//
CASE stCommand.PositionType OF
	DUT_Command_PositionType.AbsolutePosition:
		F_AddElement(_Command, _Delimiter, _ChangeTypeA);
	DUT_Command_PositionType.RelativePosition:
		F_AddElement(_Command, _Delimiter, _ChangeTypeR);
END_CASE

//
F_AddElement(_Command, _Delimiter, LREAL_TO_STRING(stCommand.Speed));

//
CASE stCommand.CoordSystem OF
	SMC_COORD_SYSTEM.ACS:
		F_AddElement(_Command, _Delimiter, _CoordSystemAcs);
	SMC_COORD_SYSTEM.MCS:
		F_AddElement(_Command, _Delimiter, _CoordSystemMcs);
	SMC_COORD_SYSTEM.PCS_1:
		F_AddElement(_Command, _Delimiter, _CoordSystemPc1);
	SMC_COORD_SYSTEM.PCS_2:
		F_AddElement(_Command, _Delimiter, _CoordSystemPc2);
	SMC_COORD_SYSTEM.TCS:
		F_AddElement(_Command, _Delimiter, _CoordSystemTcs);
	SMC_COORD_SYSTEM.WCS:
		F_AddElement(_Command, _Delimiter, _CoordSystemWcs);
	SMC_COORD_SYSTEM.ICS:
		F_AddElement(_Command, _Delimiter, _CoordSystemIcs);
END_CASE

//
CASE stCommand.CoordinateType OF
	DUT_Command_CoordinateType.Literal:
		F_AddElement(_Command, _Delimiter, _CoordTypeH);
		F_AddElement(_Command, _Delimiter, LREAL_TO_STRING(stCommand.CoordRef.X));
		F_AddElement(_Command, _Delimiter, LREAL_TO_STRING(stCommand.CoordRef.Y));
		F_AddElement(_Command, _Delimiter, LREAL_TO_STRING(stCommand.CoordRef.Z));
		F_AddElement(_Command, _Delimiter, LREAL_TO_STRING(stCommand.CoordRef.A));
		F_AddElement(_Command, _Delimiter, LREAL_TO_STRING(stCommand.CoordRef.B));
		F_AddElement(_Command, _Delimiter, LREAL_TO_STRING(stCommand.CoordRef.C));
		
	DUT_Command_CoordinateType.Variable:
		F_AddElement(_Command, _Delimiter, _CoordTypeV);
		CASE stCommand.ArrayType OF
			DUT_Command_ArrayType.StoredPosition:
				F_AddElement(_Command, _Delimiter, _ArrayTypeS);
			DUT_Command_ArrayType.VisionRegister:
				F_AddElement(_Command, _Delimiter, _ArrayTypeV);
			DUT_Command_ArrayType.Flag:
				// on damn
		END_CASE
		F_AddElement(_Command, _Delimiter, UDINT_TO_STRING(stCommand.ArrayIndex));
		
END_CASE

// only add if move type is circle
IF stCommand.MoveType = DUT_Command_MoveType.CircularMove THEN
	//
	CASE stCommand.CircleMode OF
		SMC_CIRC_MODE.BORDER:
			F_AddElement(_Command, _Delimiter, _CircleModeBor);
		SMC_CIRC_MODE.CENTER:
			F_AddElement(_Command, _Delimiter, _CircleModeCen);
		SMC_CIRC_MODE.RADIUS:
			F_AddElement(_Command, _Delimiter, _CircleModeRad);
	END_CASE
	//
	CASE stCommand.PathChoice OF
		MC_CIRC_PATHCHOICE.CLOCKWISE:
			F_AddElement(_Command, _Delimiter, _PathChoiceClw);
		MC_CIRC_PATHCHOICE.COUNTER_CLOCKWISE:
			F_AddElement(_Command, _Delimiter, _PathChoiceCcw);
	END_CASE
	//
	CASE stCommand.CircularCoordinateType OF
		DUT_Command_CoordinateType.Literal:
			F_AddElement(_Command, _Delimiter, _CoordTypeH);
			F_AddElement(_Command, _Delimiter, LREAL_TO_STRING(stCommand.CoordRef2.X));
			F_AddElement(_Command, _Delimiter, LREAL_TO_STRING(stCommand.CoordRef2.Y));
			F_AddElement(_Command, _Delimiter, LREAL_TO_STRING(stCommand.CoordRef2.Z));
			F_AddElement(_Command, _Delimiter, LREAL_TO_STRING(stCommand.CoordRef2.A));
			F_AddElement(_Command, _Delimiter, LREAL_TO_STRING(stCommand.CoordRef2.B));
			F_AddElement(_Command, _Delimiter, LREAL_TO_STRING(stCommand.CoordRef2.C));
			
		DUT_Command_CoordinateType.Variable:
			F_AddElement(_Command, _Delimiter, _CoordTypeV);
			CASE stCommand.CircularArrayType OF
				DUT_Command_ArrayType.StoredPosition:
					F_AddElement(_Command, _Delimiter, _ArrayTypeS);
				DUT_Command_ArrayType.VisionRegister:
					F_AddElement(_Command, _Delimiter, _ArrayTypeV);
				DUT_Command_ArrayType.Flag:
					// oh damn
			END_CASE
			F_AddElement(_Command, _Delimiter, UDINT_TO_STRING(stCommand.CircularArrayIndex));
			
	END_CASE

END_IF

// set function equal to command
F_BuildMoveCmd := _Command;
                  
END_FUNCTION

FUNCTION F_RoundLreal : LREAL
VAR_INPUT
   rIn : LREAL;      
   Digit: INT;         
END_VAR

VAR
   d1 : DINT;
   r0,r1,r2,Rdigit: LREAL;               
END_VAR

                    // https://forge.codesys.com/forge/talk/Engineering/thread/8d1ee86294/
rdigit   :=INT_TO_LREAL(Digit);
r0 := EXPT(10,rdigit); 
r1 := rIn * r0;
d1 := TRUNC(r1);
r2 := DINT_TO_LREAL(d1);
F_RoundLreal := r2 / r0;
                  
END_FUNCTION

FUNCTION_BLOCK FB_ParseLogicCmd
VAR_INPUT
	Command: STRING(GVL.COMMAND_LEN);
END_VAR
VAR_OUTPUT
	stCommand: ST_LogicCmd;
	Error: BOOL;
	ErrorDescription: STRING;
END_VAR
VAR
	_CmdParams: ARRAY [0..GVL.COMMAND_LEN] OF STRING;
	_i, _j, _k: INT;
END_VAR

                    // IF PASS|INPUT|REGISTER|COUNTER <index> >|<|=|>=|<= <value>
// THEN OUTPUT|JUMP|CALL|CNTUP|CNTDN|CNTRST|REGISTER|NOP <index> <value>
// ELSE OUTPUT|JUMP|CALL|CNTUP|CNTDN|CNTRST|REGISTER|NOP <index> <value>
//
// IF_Condition
// IF_Condition_Idx
// IF_Condition_Operator
// IF_Condition_Operator_Compare
// THEN_Function
// THEN_Function_Value
// THEN_Function_Idx
// ELSE_Function
// ELSE_Function_Idx
// ELSE_Function_Value

Error:=FALSE;
ErrorDescription:='';

// split command string into commands
_CmdParams:=F_SplitCmd(Command:=Command);

//
_i := 0;

// disregard the 'IF'
_i := _i + 1;

//
IF _CmdParams[_i] = TO_STRING(E_LogicIfCondition.PASS) THEN
	stCommand.IF_Condition := E_LogicIfCondition.PASS;
ELSIF  _CmdParams[_i] = TO_STRING(E_LogicIfCondition.INPUT) THEN
	stCommand.IF_Condition := E_LogicIfCondition.INPUT;
ELSIF  _CmdParams[_i] = TO_STRING(E_LogicIfCondition.REGISTER) THEN
	stCommand.IF_Condition := E_LogicIfCondition.REGISTER;
ELSIF  _CmdParams[_i] = TO_STRING(E_LogicIfCondition.COUNTER) THEN
	stCommand.IF_Condition := E_LogicIfCondition.COUNTER;
ELSIF  _CmdParams[_i] = TO_STRING(E_LogicIfCondition.FLAG) THEN
	stCommand.IF_Condition := E_LogicIfCondition.FLAG;
END_IF
_i := _i + 1;

//
IF stCommand.IF_Condition <> E_LogicIfCondition.PASS THEN
	
	//
	stCommand.IF_Condition_Idx := STRING_TO_INT(_CmdParams[_i]);
	_i := _i + 1;
	
	//
	IF _CmdParams[_i] = TO_STRING(E_LogicIfConditionOperator.GRT) THEN
		stCommand.IF_Condition_Operator := E_LogicIfConditionOperator.GRT;
	ELSIF _CmdParams[_i] = TO_STRING(E_LogicIfConditionOperator.LES) THEN
		stCommand.IF_Condition_Operator := E_LogicIfConditionOperator.LES;                   
	ELSIF _CmdParams[_i] = TO_STRING(E_LogicIfConditionOperator.EQU) THEN
		stCommand.IF_Condition_Operator := E_LogicIfConditionOperator.EQU;
	ELSIF _CmdParams[_i] = TO_STRING(E_LogicIfConditionOperator.GRE) THEN
		stCommand.IF_Condition_Operator := E_LogicIfConditionOperator.GRE;
	ELSIF _CmdParams[_i] = TO_STRING(E_LogicIfConditionOperator.LEQ) THEN
		stCommand.IF_Condition_Operator := E_LogicIfConditionOperator.LEQ;
	END_IF
	_i := _i + 1;
	
	//
	stCommand.IF_Condition_Operator_Value := STRING_TO_UDINT(_CmdParams[_i]);
	_i := _i + 1;
	
END_IF

// disregard the 'THEN'
_i := _i + 1;

//
IF _CmdParams[_i] = TO_STRING(E_LogicFunction.OUTPUT) THEN
	stCommand.THEN_Function := E_LogicFunction.OUTPUT;
ELSIF _CmdParams[_i] = TO_STRING(E_LogicFunction.JUMP) THEN
	stCommand.THEN_Function := E_LogicFunction.JUMP;
ELSIF _CmdParams[_i] = TO_STRING(E_LogicFunction.CALL) THEN
	stCommand.THEN_Function := E_LogicFunction.CALL;           
ELSIF _CmdParams[_i] = TO_STRING(E_LogicFunction.CNTUP) THEN
	stCommand.THEN_Function := E_LogicFunction.CNTUP;
ELSIF _CmdParams[_i] = TO_STRING(E_LogicFunction.CNTDN) THEN
	stCommand.THEN_Function := E_LogicFunction.CNTDN;
ELSIF _CmdParams[_i] = TO_STRING(E_LogicFunction.CNTRST) THEN
	stCommand.THEN_Function := E_LogicFunction.CNTRST;
ELSIF _CmdParams[_i] = TO_STRING(E_LogicFunction.REGISTER) THEN
	stCommand.THEN_Function := E_LogicFunction.REGISTER;
ELSIF _CmdParams[_i] = TO_STRING(E_LogicFunction.FLAG) THEN
	stCommand.THEN_Function := E_LogicFunction.FLAG;
ELSIF _CmdParams[_i] = TO_STRING(E_LogicFunction.NOP) THEN
	stCommand.THEN_Function := E_LogicFunction.NOP;
END_IF
_i := _i + 1;

//
IF stCommand.THEN_Function <> E_LogicFunction.NOP THEN
	stCommand.THEN_Function_Idx := STRING_TO_INT(_CmdParams[_i]);
	_i := _i + 1;
	IF stCommand.THEN_Function = E_LogicFunction.OUTPUT OR
		stCommand.THEN_Function = E_LogicFunction.REGISTER OR
		stCommand.THEN_Function = E_LogicFunction.FLAG THEN
			stCommand.THEN_Function_Value := STRING_TO_UDINT(_CmdParams[_i]);
			_i := _i + 1;
	END_IF
END_IF

// disregard the 'ELSE'
_i := _i + 1;

//
IF _CmdParams[_i] = TO_STRING(E_LogicFunction.OUTPUT) THEN
	stCommand.ELSE_Function := E_LogicFunction.OUTPUT;
ELSIF _CmdParams[_i] = TO_STRING(E_LogicFunction.JUMP) THEN
	stCommand.ELSE_Function := E_LogicFunction.JUMP;
ELSIF _CmdParams[_i] = TO_STRING(E_LogicFunction.CALL) THEN
	stCommand.ELSE_Function := E_LogicFunction.CALL;
ELSIF _CmdParams[_i] = TO_STRING(E_LogicFunction.CNTUP) THEN
	stCommand.ELSE_Function := E_LogicFunction.CNTUP;
ELSIF _CmdParams[_i] = TO_STRING(E_LogicFunction.CNTDN) THEN
	stCommand.ELSE_Function := E_LogicFunction.CNTDN;
ELSIF _CmdParams[_i] = TO_STRING(E_LogicFunction.CNTRST) THEN
	stCommand.ELSE_Function := E_LogicFunction.CNTRST;
ELSIF _CmdParams[_i] = TO_STRING(E_LogicFunction.REGISTER) THEN
	stCommand.ELSE_Function := E_LogicFunction.REGISTER;
ELSIF _CmdParams[_i] = TO_STRING(E_LogicFunction.FLAG) THEN
	stCommand.ELSE_Function := E_LogicFunction.FLAG;
ELSIF _CmdParams[_i] = TO_STRING(E_LogicFunction.NOP) THEN
	stCommand.ELSE_Function := E_LogicFunction.NOP;
END_IF
_i := _i + 1;

//
IF stCommand.ELSE_Function <> E_LogicFunction.NOP THEN
	stCommand.ELSE_Function_Idx := STRING_TO_INT(_CmdParams[_i]);
	_i := _i + 1;
	IF stCommand.ELSE_Function = E_LogicFunction.OUTPUT OR
		stCommand.ELSE_Function = E_LogicFunction.REGISTER OR
		stCommand.ELSE_Function = E_LogicFunction.FLAG THEN
			stCommand.ELSE_Function_Value := STRING_TO_UDINT(_CmdParams[_i]);
			_i := _i + 1;
	END_IF
END_IF
                  
END_FUNCTION_BLOCK

FUNCTION F_BuildLogicCmd : STRING(GVL.COMMAND_LEN)
VAR_INPUT
	stCommand: ST_LogicCmd;
END_VAR
VAR
    _Command: STRING(GVL.COMMAND_LEN);
END_VAR
VAR CONSTANT
	_Delimiter: STRING:=' ';
END_VAR

                    // IF PASS|INPUT|REGISTER|COUNTER <index> >|<|=|>=|<= <value>
// THEN OUTPUT|JUMP|CNTUP|CNTDN|CNTRST|REGISTER|NOP <index> <value>
// ELSE OUTPUT|JUMP|CNTUP|CNTDN|CNTRST|REGISTER|NOP <index> <value>
//
// IF_Condition
// IF_Condition_Idx
// IF_Condition_Operator
// IF_Condition_Operator_Compare
// THEN_Function
// THEN_Function_Value
// THEN_Function_Idx
// ELSE_Function
// ELSE_Function_Idx
// ELSE_Function_Value

// clear the command
_Command:='';

// build command
F_AddElement(_Command, _Delimiter, 'IF');
F_AddElement(_Command, _Delimiter, TO_STRING(stCommand.IF_Condition));
IF stCommand.IF_Condition <> E_LogicIfCondition.PASS THEN
	F_AddElement(_Command, _Delimiter, INT_TO_STRING(stCommand.IF_Condition_Idx));
	F_AddElement(_Command, _Delimiter, TO_STRING(stCommand.IF_Condition_Operator));
	F_AddElement(_Command, _Delimiter, UDINT_TO_STRING(stCommand.IF_Condition_Operator_Value));
END_IF
F_AddElement(_Command, _Delimiter, 'THEN');
F_AddElement(_Command, _Delimiter, TO_STRING(stCommand.THEN_Function));
IF stCommand.THEN_Function <> E_LogicFunction.NOP THEN
	F_AddElement(_Command, _Delimiter, INT_TO_STRING(stCommand.THEN_Function_Idx));
	IF stCommand.THEN_Function = E_LogicFunction.OUTPUT OR 
		stCommand.THEN_Function = E_LogicFunction.REGISTER OR 
		stCommand.THEN_Function = E_LogicFunction.FLAG THEN
			F_AddElement(_Command, _Delimiter, UDINT_TO_STRING(stCommand.THEN_Function_Value));
	END_IF
END_IF
IF stCommand.IF_Condition <> E_LogicIfCondition.PASS THEN
	F_AddElement(_Command, _Delimiter, 'ELSE');
	F_AddElement(_Command, _Delimiter, TO_STRING(stCommand.ELSE_Function));
	IF stCommand.ELSE_Function <> E_LogicFunction.NOP THEN
		F_AddElement(_Command, _Delimiter, INT_TO_STRING(stCommand.ELSE_Function_Idx));
		IF stCommand.ELSE_Function = E_LogicFunction.OUTPUT OR
			stCommand.ELSE_Function = E_LogicFunction.REGISTER OR
			stCommand.ELSE_Function = E_LogicFunction.FLAG THEN
				F_AddElement(_Command, _Delimiter, UDINT_TO_STRING(stCommand.ELSE_Function_Value));
		END_IF
	END_IF
END_IF

// set function equal to command
F_BuildLogicCmd := _Command;
                  
END_FUNCTION

FUNCTION F_HomeOffsetCalc : LREAL
VAR_INPUT
	CurrentOffset: LREAL;
	CurrentPosition: LREAL;
	HomeSearchDirection: MC_Direction;
END_VAR
VAR
END_VAR

                    IF HomeSearchDirection = MC_Direction.positive THEN
	F_HomeOffsetCalc := -F_RoundLreal(ABS(CurrentPosition - CurrentOffset),2);
	
ELSIF HomeSearchDirection = MC_Direction.negative THEN
	F_HomeOffsetCalc := F_RoundLreal(ABS(CurrentPosition - CurrentOffset),2);
	
ELSE
	F_HomeOffsetCalc := CurrentOffset;
	
END_IF
                  
END_FUNCTION

FUNCTION_BLOCK FB_ProgramProcessor EXTENDS FB_Module
VAR_IN_OUT
	Programs: ARRAY [GVL.PROG_ARR_BEG..GVL.PROG_ARR_END] OF DUT_Program;
	J1, J2, J3, J4, J5, J6: AXIS_REF_SM3;
	AxisGroup: AXIS_GROUP_REF_SM3;
	GroupHandler: FB_GroupHandler;
	CmdIO: ST_LogicCmdIO;
END_VAR
VAR_INPUT
	Enable: BOOL;
END_VAR
VAR_OUTPUT
	ItfActiveProcessorUnitMode	: PACK_ML.IUnitMode;
	ItfActiveModule: ItfModule;
	StatusText: STRING(255);
    GCodeLines: ARRAY[0..SMC_GCodeViewer.c_uiLines] OF STRING;
END_VAR
VAR
	_DummyUnitMode: PACK_ML.UnitMode;
	_UnitModeCurrentState: PACK_ML.State;
	_Returning:  ARRAY [GVL.PROG_ARR_BEG..GVL.PROG_ARR_END] OF BOOL;
	_ReturnPrograms: ARRAY [GVL.PROG_ARR_BEG..GVL.PROG_ARR_END] OF UINT;
	_ReturnCommands: ARRAY [GVL.PROG_CMDS_ARR_BEG..GVL.PROG_CMDS_ARR_END + 1] OF UINT; // +1 because we want to be able to tell if calling program was on last command
	_CurrentPrgIdx: UINT;
	_ProcessCommands: FB_CommandProcessor;
	_Commands: ARRAY [GVL.PROG_CMDS_ARR_BEG..GVL.PROG_CMDS_ARR_END] OF DUT_Command;
    _ErrorRtrig: R_TRIG;
	_i, _j, _k: INT;
	_FirstScan: BOOL:=TRUE;
END_VAR

VAR CONSTANT
	_STEP_DONE: 			INT := 1000;
	_STEP_IDLE: 			INT := 0000;
	_STEP_PRG:				INT := 0010;
	_STEP_WAIT_EXECUTE:		INT := 0020;
	_STEP_WAIT_IDLE:		INT := 0025;
	_STEP_ERR:              INT := 0030;
END_VAR

                    //
SUPER^();

//
IF _FirstScan THEN
	// will exception if we don't set this on first scan
	_DummyUnitMode(sName := 'Active Processor', 
					eInitialState := PACK_ML.State.Idle,
					xActive := TRUE);
	ItfActiveProcessorUnitMode := _DummyUnitMode;
END_IF

// this is at best a hack and needs to be rethought out.
// we logically cant assign a process as the active unit mode 
// at start up so we use this dummy one
CASE _DummyUnitMode.CurrentState OF
	PACK_ML.State.Stopped,
	PACK_ML.State.Aborted,
	PACK_ML.State.Held,
	PACK_ML.State.Suspended,
	PACK_ML.State.Complete,
	PACK_ML.State.Idle:
		//
	PACK_ML.State.Resetting,
	PACK_ML.State.Starting,
	PACK_ML.State.Execute,
	PACK_ML.State.Suspending,
	PACK_ML.State.UnSuspending,
	PACK_ML.State.Holding,
	PACK_ML.State.UnHolding,
	PACK_ML.State.Completing,
	PACK_ML.State.Aborting,
	PACK_ML.State.Stopping,
	PACK_ML.State.Clearing:
		_DummyUnitMode.ActingStateCompleted();
END_CASE

// PackML state machine implementation
_UnitModeCurrentState := SUPER^._UnitMode.CurrentState;

//
_ErrorRtrig(CLK:=_ProcessCommands.Error);
IF _ErrorRtrig.Q THEN
	SUPER^.M_Error(Description:=CONCAT('Command Processor Error: ', _ProcessCommands.ErrorDescription));
	StatusText:=SUPER^.ErrorDescription;
END_IF

//
_ProcessCommands(
	StoredPositions:=SUPER^.StoredPositions,
	VisionRegisters:=SUPER^.VisionRegisters,
	Flags:=SUPER^.Flags,
	J1:=J1, J2:=J2, J3:=J3, J4:=J4, J5:=J5, J6:=J6,
	AxisGroup:= AxisGroup,
	GroupHandler:= GroupHandler,
	CmdIO:=CmdIO,
	PrgProcessor:= THIS^,
    GCodeLines => GCodeLines,
	Enable:= Enable,
	Error=> ,
	StatusText=>StatusText);	

_FirstScan := FALSE;
                  

METHOD PUBLIC M_CallProgram : bool
VAR_INPUT
	ProgramNumber: UINT; // program to call
	ReturnProgram: UINT; // number of the program to return to when the call program ends
	ReturnCommand: UINT; // number of the command to start from when called program ends
END_VAR
                          {warning disable C0371}
IF ProgramNumber <= GVL.PROG_ARR_END AND_THEN ProgramNumber >= GVL.PROG_ARR_BEG
	AND_THEN ReturnProgram <= GVL.PROG_ARR_END AND_THEN ReturnProgram >= GVL.PROG_ARR_BEG
	AND_THEN SUPER^.PropCurrentState = PACK_ML.State.Execute THEN
		IF _ProcessCommands.M_SetCommands(StartingCommand:=0, Commands:=Programs[ProgramNumber].Commands) THEN
			IF ReturnCommand <= GVL.PROG_CMDS_ARR_END + 1 AND_THEN ReturnCommand >= GVL.PROG_CMDS_ARR_BEG THEN // +1 because we want to be able to tell if calling program was on last command
				_Returning[ProgramNumber] := TRUE;
				_ReturnPrograms[ProgramNumber] := ReturnProgram;
				_ReturnCommands[ProgramNumber] := ReturnCommand;
			END_IF
			_CurrentPrgIdx := ProgramNumber;
			M_CallProgram := TRUE;
		ELSE
			M_CallProgram := FALSE;
		END_IF
ELSE
	M_CallProgram := FALSE;
END_IF
{warning restore C0371}
                        
END_METHOD

METHOD PROTECTED M_Complete : BOOL
                          // once complete, reset to get back to idle
SUPER^._UnitMode.Reset();
                        
END_METHOD

METHOD PROTECTED M_Resetting : BOOL
                          CASE _SeqResetting OF
	0:
		_ProcessCommands.M_Home();
		_SeqResetting := _SeqResetting + 1;
	1:
		IF _ProcessCommands.PropCurrentState = PACK_ML.State.Idle THEN
			_SeqResetting := 0;
			SUPER^.M_StateComplete();
		END_IF
		
END_CASE

SUPER^.M_Reset();

(*IF ItfActiveModule <> 0 THEN
	CASE _Seq OF
		0:
			IF NOT ItfActiveModule.PropCurrentState = PACK_ML.State.Idle THEN
				ItfActiveModule.M_Home();
				_Seq := 1;
			ELSE
				SUPER^.M_StateComplete();
			END_IF
		1:
			IF ItfActiveModule.PropCurrentState = PACK_ML.State.Idle THEN
				_Seq := 0;
			END_IF
			
	END_CASE
	
ELSE
	SUPER^.M_StateComplete();
	_Seq := 0;
	
END_IF*)
                        
END_METHOD

METHOD PROTECTED M_Idle : BOOL
                          // in this state, we want to reset all the function blocks and hang out
FOR _i:=GVL.PROG_ARR_BEG TO GVL.PROG_ARR_END BY 1 DO
	_Returning[_i] := FALSE;
END_FOR
(*FOR _i:=GVL.PROG_ARR_BEG TO GVL.PROG_ARR_END BY 1 DO
	_ReturnPrograms[_i] := 0;
END_FOR
FOR _i:=GVL.PROG_CMDS_ARR_BEG TO GVL.PROG_CMDS_ARR_END BY 1 DO
	_ReturnCommands[_i] := 0;
END_FOR*)
_SeqMain := _STEP_IDLE;
_SeqAborting := 0;
_SeqClearing := 0;
_SeqResetting := 0;
                        
END_METHOD

METHOD PROTECTED M_SetPackML : BOOL
                          // SUPER already does this but the default is eInitialState:=PACK_ML.State.Idle 
// and we want PACK_ML.State.Aborted for the Orchestrator
SUPER^._UnitMode(sName := 'Program Processor',
				eInitialState := PACK_ML.State.Aborted,
				xActive := TRUE);
                        
END_METHOD

METHOD PROTECTED M_Starting : BOOL
                          // here we want to clear things and get ready for the execute state
// we can consider this the "INIT" state
(*FOR _i:=GVL.PROG_ARR_BEG TO GVL.PROG_ARR_END BY 1 DO
	_Returning[_i] := FALSE;
END_FOR
FOR _i:=GVL.PROG_ARR_BEG TO GVL.PROG_ARR_END BY 1 DO
	_ReturnPrograms[_i] := 0;
END_FOR
FOR _i:=GVL.PROG_CMDS_ARR_BEG TO GVL.PROG_CMDS_ARR_END BY 1 DO
	_ReturnCommands[_i] := 0;
END_FOR*)
//_CurrentPrgIdx := 0;
_SeqMain := _STEP_PRG;
SUPER^.M_StateComplete();
                        
END_METHOD

METHOD PROTECTED M_Execute : BOOL
VAR
    _ErrorDescription: STRING;
END_VAR
                          {warning disable C0371}
// here we want to execute our commands/jobs/etc and set completed when done.
//
CASE _SeqMain OF
  	_STEP_DONE:
		_SeqMain := _STEP_IDLE;
		
	_STEP_IDLE:
		// hang out here until called to run
		_CurrentPrgIdx := 0;
		SUPER^.M_StateComplete();
		
	_STEP_PRG: //
		IF NOT Enable THEN
			_SeqMain := _STEP_DONE;
            IF NOT GVL.Enable THEN
                _ErrorDescription := 'Robot not enabled';
            END_IF
            IF NOT PersistentVars.Flags[GVL.HOME_COMPLETE].Value THEN
                _ErrorDescription := CONCAT(_ErrorDescription, ' | Robot not homed');
            END_IF
            IF GVL.xActiveAlarm THEN
                _ErrorDescription := CONCAT(_ErrorDescription, ' | Active alarms exist');
            END_IF
            IF _ErrorDescription = '' THEN
                _ErrorDescription := 'Not enabled';
            END_IF
            _M_Error(Description := _ErrorDescription);
            
		ELSIF _CurrentPrgIdx <= GVL.PROG_ARR_END AND _CurrentPrgIdx >= GVL.PROG_ARR_BEG THEN
			//
			StatusText := '';
			ItfActiveModule := _ProcessCommands;
			ItfActiveProcessorUnitMode := _ProcessCommands.ItfUnitMode;
			
			IF _ProcessCommands.M_SetCommands(StartingCommand:=0, Commands:=Programs[_CurrentPrgIdx].Commands) THEN
				_ProcessCommands.M_Start();
				_SeqMain := _STEP_WAIT_EXECUTE;
			ELSE
				SUPER^.M_Error('Failed to set Command Processor. Check commands.');
				_SeqMain := _STEP_ERR;
			END_IF
			
				
		ELSE
			_SeqMain := _STEP_DONE;
		END_IF
		
	_STEP_WAIT_EXECUTE:
		IF _ProcessCommands.PropCurrentState = PACK_ML.State.Execute THEN
			_SeqMain := _STEP_WAIT_IDLE;
		END_IF
		
	_STEP_WAIT_IDLE: // wait for program to finish
		//
		IF _ProcessCommands.PropCurrentState = PACK_ML.State.Idle THEN
			IF _Returning[_CurrentPrgIdx] THEN
				_Returning[_CurrentPrgIdx] := FALSE;
				IF _ReturnPrograms[_CurrentPrgIdx] <= GVL.PROG_ARR_END AND_THEN _ReturnPrograms[_CurrentPrgIdx] >= GVL.PROG_ARR_BEG
					AND_THEN _ReturnCommands[_CurrentPrgIdx] <= GVL.PROG_CMDS_ARR_END + 1 AND_THEN _ReturnCommands[_CurrentPrgIdx] >= GVL.PROG_CMDS_ARR_BEG // +1 because we want to be able to tell if calling program was on last command
					THEN
						//
						IF _ProcessCommands.M_SetCommands(StartingCommand:=_ReturnCommands[_CurrentPrgIdx], Commands:=Programs[_ReturnPrograms[_CurrentPrgIdx]].Commands) THEN
							_CurrentPrgIdx := _ReturnPrograms[_CurrentPrgIdx];
							_ProcessCommands.M_Start();
							_SeqMain := _STEP_WAIT_EXECUTE;
						ELSE
							SUPER^.M_Error('Failed to set Command Processor. Check commands.');
							_SeqMain := _STEP_ERR;
						END_IF
				ELSE
					_SeqMain := _STEP_DONE;
				END_IF
			ELSE
				_SeqMain := _STEP_DONE;
			END_IF
		END_IF
		//
		IF _ProcessCommands.PropError THEN
			SUPER^._UnitMode.Suspend();
			_SeqMain := _STEP_ERR;
		END_IF
		
	_STEP_ERR: //
	
END_CASE

// watch for rising edge of idle state. this was done for all processors since 
// the vision processor runs in a separate task and isnt guaranteed to start in the same 
// PLC scan.
//_ProcessorDoneRtrig(clk:=ItfActiveProcessorUnitMode.CurrentState = PACK_ML.State.Idle);
{warning restore C0371}
                        
END_METHOD

METHOD PROTECTED M_Suspending : BOOL
                          IF ItfActiveModule <> 0 THEN
	IF ItfActiveModule.PropCurrentState = PACK_ML.State.Execute THEN
		ItfActiveModule.M_Hold();
		IF ItfActiveModule.PropCurrentState = PACK_ML.State.Held THEN
			SUPER^.M_StateComplete();
		END_IF
	ELSE
		SUPER^.M_StateComplete();
	END_IF
	
ELSE
	SUPER^.M_StateComplete();
	
END_IF
                        
END_METHOD

METHOD PROTECTED M_UnSuspending : BOOL
                          //
IF ItfActiveModule <> 0 THEN
	ItfActiveModule.M_Start();
	IF ItfActiveModule.PropCurrentState = PACK_ML.State.Execute THEN
		SUPER^.M_StateComplete();
	END_IF
	
ELSE
	SUPER^.M_StateComplete();
	
END_IF

//
_SeqMain := _STEP_WAIT_IDLE;
                        
END_METHOD

METHOD PROTECTED M_Holding : BOOL
                          IF ItfActiveModule <> 0 THEN
	ItfActiveModule.M_Hold();
	IF ItfActiveModule.PropCurrentState = PACK_ML.State.Held THEN
		SUPER^.M_StateComplete();
	END_IF
ELSE
	SUPER^.M_StateComplete();
END_IF
                        
END_METHOD

METHOD PROTECTED M_Unholding : BOOL
                          //
IF ItfActiveModule <> 0 THEN
	ItfActiveModule.M_Start();
	IF ItfActiveModule.PropCurrentState = PACK_ML.State.Execute THEN
		SUPER^.M_StateComplete();
	END_IF
	
ELSE
	SUPER^.M_StateComplete();
	
END_IF

//
_SeqMain := _STEP_WAIT_IDLE;
                        
END_METHOD

METHOD PROTECTED M_Aborting : BOOL
                          CASE _SeqAborting OF
	0:
		_ProcessCommands.M_Abort();
		_SeqAborting := _SeqAborting + 1;
	1:
		IF _ProcessCommands.PropCurrentState = PACK_ML.State.Aborted THEN
			_SeqAborting := 0;
			SUPER^.M_StateComplete();
		END_IF
		
END_CASE

(*IF ItfActiveModule <> 0 THEN
	ItfActiveModule.M_Abort();
	IF ItfActiveModule.PropCurrentState = PACK_ML.State.Aborted THEN
		SUPER^.M_StateComplete();
	END_IF
ELSE
	SUPER^.M_StateComplete();
END_IF*)
                        
END_METHOD

METHOD PROTECTED M_Stopping : BOOL
                          IF ItfActiveModule <> 0 THEN
	ItfActiveModule.M_Stop();
	IF ItfActiveModule.PropCurrentState = PACK_ML.State.Idle 
		OR ItfActiveModule.PropCurrentState = PACK_ML.State.Stopped 
		OR ItfActiveModule.PropCurrentState = PACK_ML.State.Aborted 
		OR ItfActiveModule.PropCurrentState = PACK_ML.State.Complete THEN
			SUPER^.M_StateComplete();
	END_IF
	
ELSE
	SUPER^.M_StateComplete();
	
END_IF
                        
END_METHOD

METHOD PROTECTED M_Clearing : BOOL
                          SUPER^.M_StateComplete();

(*IF SUPER^.Flags[GVL.HOME_COMPLETE].Value THEN
	CASE _SeqClearing OF
		0:
			_ProcessMoveCommand.M_Home();
			_SeqClearing := _SeqClearing + 1;
		1:
			IF _ProcessMoveCommand.PropCurrentState = PACK_ML.State.Idle THEN
				_SeqClearing := _SeqClearing + 1;
			END_IF
		2:
			IF NOT _ProcessMoveCommand.Error THEN
				_ProcessMoveCommand.Command := GVL.Pose2;
				_ProcessMoveCommand.M_Start();
				_SeqClearing := _SeqClearing + 1;
			ELSE
				SUPER^._M_Error(Description:='Move processor errored. Please reset and try again');
				_SeqClearing := -1;
			END_IF
		3:
			IF _ProcessMoveCommand.PropCurrentState = PACK_ML.State.Execute THEN
				_SeqClearing := _SeqClearing + 1;
			END_IF
		4:
			IF _ProcessMoveCommand.PropCurrentState = PACK_ML.State.Complete 
				OR _ProcessMoveCommand.PropCurrentState = PACK_ML.State.Stopped 
				OR _ProcessMoveCommand.PropCurrentState = PACK_ML.State.Aborted
				OR _ProcessMoveCommand.PropCurrentState = PACK_ML.State.Idle  THEN
					SUPER^.M_StateComplete();
					_SeqClearing := 0;
			END_IF
	END_CASE
ELSE
	SUPER^._M_Error(Description:='Drives are not homed. Please home and try again');
	_SeqClearing := -1;
END_IF

IF _ProcessMoveCommand.Error THEN
	SUPER^._M_Error(Description:='Move processor in error state. Please reset and try again');
	_SeqClearing := -1;
END_IF
*)

(*
IF ItfActiveModule <> 0 THEN
	//
	CASE _Seq OF
		0:
			IF NOT ItfActiveModule.PropCurrentState = PACK_ML.State.Stopped THEN
				ItfActiveModule.M_Abort();
				_Seq := 1;
			ELSE
				SUPER^.M_StateComplete();
			END_IF
		1:
			CASE ItfActiveModule.PropCurrentState OF
				PACK_ML.State.Aborted:
					ItfActiveModule.Clear();
				PACK_ML.State.Stopped:
					_Seq := 0;
			END_CASE
			
	END_CASE
ELSE
	_Seq := 0;
	SUPER^.M_StateComplete();
END_IF
*)

                        
END_METHOD

METHOD PUBLIC M_SetProgram : BOOL
VAR_INPUT
	ProgramNumber: UINT;
END_VAR
                          IF ProgramNumber >= GVL.PROG_ARR_BEG AND ProgramNumber <= GVL.PROG_ARR_END THEN
	_CurrentPrgIdx := ProgramNumber;
	M_SetProgram := TRUE;
ELSE
	M_SetProgram := FALSE;
END_IF
                        
END_METHOD

METHOD PRIVATE _M_Error
VAR_INPUT
    Description: STRING;
END_VAR
                          SUPER^.M_Error(Description := CONCAT('Program Processor: ', Description));
                        
END_METHOD

{attribute 'monitoring' := 'variable'}
PROPERTY PUBLIC P_CurrentProgram : REFERENCE TO UINT
GET
VAR
END_VAR
                            P_CurrentProgram REF= _CurrentPrgIdx;
                          
END_GET
END_PROPERTY

{attribute 'monitoring' := 'variable'}
PROPERTY PUBLIC P_CurrentCommand : REFERENCE TO DUT_Command
GET
VAR
END_VAR
                            P_CurrentCommand REF= _ProcessCommands.P_CurrentCommand;
                          
END_GET
END_PROPERTY

{attribute 'monitoring' := 'variable'}
PROPERTY PUBLIC P_CurrentCommandIndex : REFERENCE TO UINT
GET
VAR
END_VAR
                            P_CurrentCommandIndex REF= _ProcessCommands.P_CurrentCommandIndex;
                          
END_GET
END_PROPERTY
END_FUNCTION_BLOCK

FUNCTION_BLOCK FB_Controller EXTENDS FB_PythonServerHandler
VAR_INPUT
END_VAR
VAR_OUTPUT
END_VAR
VAR
	Controller: ST_Controller;
	ControllerStates: ARRAY [0..254] OF BYTE;
	ControllerStatesTemp: ARRAY [0..254] OF BYTE;
	ReadStringTemp: STRING(255);
	RecordLast: DINT;
	ReconnectTimer: TON:=(PT:=T#5S);
	
	_SetColor: BOOL;
	_Red: INT:=0;
	_Green: INT:=255;
	_Blue: INT:=0;
	
	_SetMicrophoneState: BOOL;
	_MicrophoneState: BOOL;
	
	_SetPlayerID: BOOL;
	_PlayerID: E_ControllerPlayerID;
	
	_SetBrightness: BOOL;
	_Brightness: E_ControllerBrightness;
	
	_SetMotorIntensity: BOOL;
	_Motor: E_ControllerMotor;
	_MotorIntensity: USINT; // 0-255
	_MotorIntensityDuration: REAL; // ms
	
	_SetTriggerMode: BOOL;
	_TriggerModeTrigger: E_ControllerTrigger;
	_TriggerModeMode: E_ControllerTriggerMode;
	
	_SetTriggerForce: BOOL;
	_TriggerForceTrigger: E_ControllerTrigger;
	_TriggerForceParameter: E_ControllerTriggerForceParameter;
	_TriggerForceIntensity: USINT;
	
	_i, _j, _k: INT;
	FirstScan: BOOL:=TRUE;
END_VAR
VAR CONSTANT
	States: STRING:='states: ';
END_VAR

                    SUPER^();

// copy over controller states when a new message is received
IF SUPER^.P_RecordNumber <> RecordLast THEN
	RecordLast := SUPER^.P_RecordNumber;
	IF FIND(SUPER^.P_RawReadString, States) > 0 THEN // TODO this is getting messy. need to overhaul how this works
		ControllerStatesTemp := SUPER^.P_RawReadByteArray;
		FOR _i:=0 TO UINT_TO_INT(SIZEOF(ControllerStates)) - LEN(States) BY 1 DO
			ControllerStates[_i] := ControllerStatesTemp[_i + LEN(States)];
		END_FOR
		
	END_IF
END_IF

//
_M_EvaluateControllerStates(States:=ControllerStates);
_M_SetColor();
_M_SetMicrophoneState();
_M_SetPlayerID();
_M_SetBrightness();
_M_SetMotorIntensity();
_M_SetTriggerMode();
_M_SetTriggerForce();

// try to reconnect to the server when data stops?
// leave this commented out until we have a better condition
// the edge case is when the controller is connected via bluetooth 
// but for some reason the server is not connected to it.
// maybe work this issue out on the server side.
(*ReconnectTimer(IN:= RecordLast=SUPER^.P_RecordNumber);
IF ReconnectTimer.Q THEN
	ReconnectTimer(IN:=FALSE);
	SUPER^.M_Reconnect();
END_IF*)

FirstScan:=FALSE;
                  

METHOD PRIVATE _M_EvaluateControllerStates : BOOL
VAR_INPUT
	States: ARRAY[0..254] OF BYTE;
END_VAR
VAR_STAT
	_i, _j, _k: UINT;
	_FirstScan: BOOL:=TRUE;
	_HeartbeatTimer: TON:=(PT:=T#2S);
	_Heartbeat: USINT:=0;
	_HeartbeatLast: USINT:=0;
END_VAR
VAR CONSTANT
END_VAR
                          IF _FirstScan THEN
	//
END_IF

//
_Heartbeat := States[0] OR States[7]; // States[0] appears to be bluetooth and States[7] appears to be wired
IF _Heartbeat <> _HeartbeatLast THEN
	_HeartbeatLast := _Heartbeat;
	_HeartbeatTimer(IN:=FALSE);
ELSE
	_HeartbeatTimer(IN:=TRUE);
END_IF
Controller.Connected S= NOT _HeartbeatTimer.IN;
Controller.Connected R= _HeartbeatTimer.Q;

// clear all the data if the controller disconnects
IF NOT Controller.Connected THEN
	//MemUtils.MemSet(pbyBuffer:=ADR(States), byValue:=0, dwSize:=SIZEOF(States)); 
	FOR _i:=1 TO 254 BY 1 DO // start at 1 so we dont overwrite the heartbeat
		States[_i] := 0;
	END_FOR
END_IF

Controller.Joysticks.Left.X					:= States[1];
Controller.Joysticks.Left.Y					:= States[2];
Controller.Joysticks.Right.X				:= States[3];
Controller.Joysticks.Right.Y				:= States[4];
Controller.Triggers.Left.Two				:= States[5];
Controller.Triggers.Right.Two				:= States[6];

//UNUSED									:= States[7];

Controller.Buttons.Triangle 				:= States[8].7;
Controller.Buttons.Circle 					:= States[8].6;
Controller.Buttons.Cross 					:= States[8].5;
Controller.Buttons.Square 					:= States[8].4;
Controller.Dpad								:= F_DpadState(States[8] AND 16#0F);

Controller.Joysticks.Right.ThreeButton 		:= States[9].7;
Controller.Joysticks.Left.ThreeButton 		:= States[9].6;
Controller.Buttons.Options 					:= States[9].5;
Controller.Buttons.Share 					:= States[9].4;
Controller.Triggers.Right.TwoButton 		:= States[9].3;
Controller.Triggers.Left.TwoButton 			:= States[9].2;
Controller.Triggers.Right.One 				:= States[9].1;
Controller.Triggers.Left.One 				:= States[9].0;

Controller.Buttons.PS						:= States[10].0;
Controller.Buttons.Touch					:= States[10].1;
Controller.Buttons.Mic						:= States[10].2;

//UNUSED									:= States[11];
//UNUSED									:= States[12];
//UNUSED									:= States[13];
//UNUSED									:= States[14];
//UNUSED									:= States[15];

{warning disable C0308}
Controller.Accelerometer.X					:= SHL(States[16], 8) OR States[17];
Controller.Accelerometer.Y					:= SHL(States[18], 8) OR States[19];
Controller.Accelerometer.Z					:= SHL(States[20], 8) OR States[21];

Controller.Gyroscope.Pitch					:= SHL(States[22], 8) OR States[23];
Controller.Gyroscope.Yaw					:= SHL(States[24], 8) OR States[25];
Controller.Gyroscope.Roll					:= SHL(States[26], 8) OR States[27];

//UNUSED									:= States[28];
//UNUSED									:= States[29];
//UNUSED									:= States[30];
//UNUSED									:= States[31];
//UNUSED									:= States[32];

Controller.Trackpads.One.ID					:= States[33] AND 16#7F;
Controller.Trackpads.One.Active				:= (States[33] AND 16#80) = 0;
Controller.Trackpads.One.X					:= SHL((States[35] AND 16#0F), 8) OR States[34];
Controller.Trackpads.One.Y					:= SHL(States[36], 4) OR SHR((States[35] AND 16#F0), 4);
Controller.Trackpads.Two.ID					:= States[37] AND 16#7F;
Controller.Trackpads.Two.Active				:= (States[37] AND 16#80) = 0;
Controller.Trackpads.Two.X					:= SHL((States[39] AND 16#0F), 8) OR States[38];
Controller.Trackpads.Two.Y					:= SHL(States[40], 4) OR SHR((States[39] AND 16#F0), 4);
{warning restore C0308}

//UNUSED									:= States[41];
//UNUSED									:= States[42];
//UNUSED									:= States[43];
//UNUSED									:= States[44];
//UNUSED									:= States[45];
//UNUSED									:= States[46];
//UNUSED									:= States[47];
//UNUSED									:= States[48];
//UNUSED									:= States[49];
//UNUSED									:= States[50];
//UNUSED									:= States[51];
//UNUSED									:= States[52];

// from kit-nya
Controller.Battery.State					:= SHR(States[53] AND 16#F0, 4);
Controller.Battery.Level					:= MIN((States[53] AND 16#0F) * 10 + 5, 100); // TODO this will show a value of 5 when controller is disconnected.

// dont put anything below this
_FirstScan := FALSE;
                        
END_METHOD

METHOD PUBLIC M_SetColor : BOOL
VAR_INPUT
	Red: INT:=0;
	Green: INT:=255;
	Blue: INT:=0;
END_VAR
                          IF Red>=0 AND_THEN Red<=255
	AND_THEN Green>=0 AND_THEN Green<=255
	AND_THEN Blue>=0 AND_THEN Blue<=255THEN
		M_SetColor := TRUE;
		_SetColor:=TRUE;
		_Red:=Red;
		_Green:=Green;
		_Blue:=Blue;
ELSE
	M_SetColor := FALSE;
END_IF
                        
END_METHOD

METHOD PUBLIC M_SetPlayerID : BOOL
VAR_INPUT
	PlayerID: E_ControllerPlayerID;
END_VAR
                          M_SetPlayerID := TRUE;
_PlayerID := PlayerID;
_SetPlayerID := TRUE;

                        
END_METHOD

METHOD PUBLIC M_SetMicrophoneState : BOOL
VAR_INPUT
	State: BOOL;
END_VAR
                          M_SetMicrophoneState := TRUE;
_MicrophoneState := State;
_SetMicrophoneState := TRUE;
                        
END_METHOD

METHOD PRIVATE _M_SetColor : BOOL
VAR_INPUT
END_VAR
VAR
	_Command: STRING(255);
END_VAR
                          IF NOT SUPER^._Busy AND_THEN _SetColor THEN
	_SetColor := FALSE;
	
	_Command := CONCAT('cmd: setColorI:', INT_TO_STRING(_Red));
	_Command := CONCAT(_Command, ',');
	_Command := CONCAT(_Command, INT_TO_STRING(_Green));
	_Command := CONCAT(_Command, ',');
	_Command := CONCAT(_Command, INT_TO_STRING(_Blue));
	
	SUPER^._M_Execute(Command:=_Command, Timeout:=5);
	SUPER^(); // call super here so other methods see it busy.
END_IF
                        
END_METHOD

METHOD PRIVATE _M_SetMicrophoneState : BOOL
VAR_INPUT
END_VAR
VAR
	_Command: STRING(255);
END_VAR
                          IF NOT SUPER^._Busy AND _SetMicrophoneState THEN
	_SetMicrophoneState := FALSE;
	
	_Command := CONCAT('cmd: setMicrophoneState:', BOOL_TO_STRING(_MicrophoneState));
	
	SUPER^._M_Execute(Command:=_Command, Timeout:=5);
	SUPER^(); // call super here so other methods see it busy.
END_IF;
                        
END_METHOD

METHOD PRIVATE _M_SetPlayerID : BOOL
VAR_INPUT
END_VAR
VAR
	_Command: STRING(255);
END_VAR
                          IF NOT SUPER^._Busy AND _SetPlayerID THEN
	_SetPlayerID := FALSE;
	
	_Command := CONCAT('cmd: setPlayerID:', INT_TO_STRING(_PlayerID));
	
	SUPER^._M_Execute(Command:=_Command, Timeout:=5);
	SUPER^(); // call super here so other methods see it busy.
END_IF
                        
END_METHOD

METHOD PRIVATE _M_SetBrightness : BOOL
VAR_INPUT
END_VAR
                          IF NOT SUPER^._Busy AND _SetBrightness THEN
	_SetBrightness := FALSE;
	
	_Command := CONCAT('cmd: setBrightness:', INT_TO_STRING(_Brightness));
	
	SUPER^._M_Execute(Command:=_Command, Timeout:=5);
	SUPER^(); // call super here so other methods see it busy.
END_IF
                        
END_METHOD

METHOD PUBLIC M_SetBrightness : BOOL
VAR_INPUT
	Brightness: E_ControllerBrightness;
END_VAR
                          M_SetBrightness := TRUE;
_Brightness := Brightness;
_SetBrightness := TRUE;
                        
END_METHOD

METHOD PUBLIC M_SetMotorIntensity : BOOL
VAR_INPUT
	Motor: E_ControllerMotor;
	Intensity: USINT; // 0-255
	Duration: REAL; // s
END_VAR
                          IF Intensity >=0 AND_THEN Intensity <= 255 AND_THEN Duration <= 5000 THEN
	M_SetMotorIntensity := TRUE;
	_SetMotorIntensity := TRUE;
	_Motor := Motor;
	_MotorIntensity := Intensity;
	_MotorIntensityDuration := Duration;
ELSE
	M_SetMotorIntensity := FALSE;
END_IF
                        
END_METHOD

METHOD PRIVATE _M_SetMotorIntensity : BOOL
VAR_INPUT
END_VAR
VAR
	_Command: STRING(255);
END_VAR
                          IF NOT SUPER^._Busy AND _SetMotorIntensity THEN
	_SetMotorIntensity := FALSE;
	
	IF _Motor = E_ControllerMotor.Left THEN
		_Command := 'cmd: setLeftMotor:';
	ELSE
		_Command := 'cmd: setRightMotor:';
	END_IF
	_Command := CONCAT(_Command, USINT_TO_STRING(_MotorIntensity));
	_Command := CONCAT(_Command, ',');
	_Command := CONCAT(_Command, REAL_TO_STRING(_MotorIntensityDuration));
	
	SUPER^._M_Execute(Command:=_Command, Timeout:=5);
	SUPER^(); // call super here so other methods see it busy.
END_IF
                        
END_METHOD

METHOD PRIVATE _M_SetTriggerMode : BOOL
VAR_INPUT
END_VAR
VAR
	_Command: STRING(255);
END_VAR
                          
IF NOT SUPER^._Busy AND _SetTriggerMode THEN
	_SetTriggerMode := FALSE;
	
	IF _TriggerModeTrigger = E_ControllerTrigger.Left THEN
		_Command := 'cmd: setLeftTriggerMode:';
	ELSE
		_Command := 'cmd: setRightTriggerMode:';
	END_IF
	_Command := CONCAT(_Command, INT_TO_STRING(_TriggerModeMode));
	
	SUPER^._M_Execute(Command:=_Command, Timeout:=5);
	SUPER^(); // call super here so other methods see it busy.
END_IF
                        
END_METHOD

METHOD PUBLIC M_SetTriggerMode : BOOL
VAR_INPUT
	Trigger: E_ControllerTrigger;
	Mode: E_ControllerTriggerMode;
END_VAR
                          M_SetTriggerMode := TRUE;
_SetTriggerMode := TRUE;
_TriggerModeTrigger := Trigger;
_TriggerModeMode := Mode;
                        
END_METHOD

METHOD PRIVATE _M_SetTriggerForce : BOOL
VAR_INPUT
END_VAR
VAR
	_Command: STRING(255);
END_VAR
                          
IF NOT SUPER^._Busy AND _SetTriggerForce THEN
	_SetTriggerForce := FALSE;
	
	IF _TriggerForceTrigger = E_ControllerTrigger.Left THEN
		_Command := 'cmd: setLeftTriggerForce:';
	ELSE
		_Command := 'cmd: setRightTriggerForce:';
	END_IF
	_Command := CONCAT(_Command, INT_TO_STRING(_TriggerForceParameter));
	_Command := CONCAT(_Command, ',');
	_Command := CONCAT(_Command, USINT_TO_STRING(_TriggerForceIntensity));
	
	SUPER^._M_Execute(Command:=_Command, Timeout:=5);
	SUPER^(); // call super here so other methods see it busy.
END_IF
                        
END_METHOD

METHOD PUBLIC M_SetTriggerForce : BOOL
VAR_INPUT
	Trigger: E_ControllerTrigger;
	Parameter: E_ControllerTriggerForceParameter;
	Intensity: USINT; // 0-255
END_VAR
                          IF Intensity >= 0 AND Intensity <= 255 THEN
	M_SetTriggerForce := TRUE;
	_SetTriggerForce:=TRUE;
	_TriggerForceTrigger := Trigger;
	_TriggerForceParameter := Parameter;
	_TriggerForceIntensity := Intensity;
ELSE
	M_SetTriggerForce := FALSE;
END_IF
                        
END_METHOD

{attribute 'monitoring' := 'variable'}
PROPERTY PUBLIC P_State : REFERENCE TO ST_Controller
GET
VAR
END_VAR
                            P_State REF= Controller;
                          
END_GET
END_PROPERTY
END_FUNCTION_BLOCK

FUNCTION_BLOCK FB_PythonServerHandler
VAR_INPUT
	sIpAddress: STRING(19):='127.0.0.1';
	uPort: UINT:=50011;
END_VAR
VAR_OUTPUT
END_VAR
VAR
	_Done: BOOL;
	_Busy: BOOL;
	_Error: BOOL;
	_ErrorDescription: STRING;
	_Response: STRING(255);
	_WorkerUid: STRING;
	_Execute: BOOL;
	_Reset: BOOL:=FALSE;
	_ResetRtrig: R_TRIG;
	_Step: INT;
	_Command: STRING(255);
	_ReadRecordLast: DINT;
	_TcpClient: FB_TcpClient;
	_TimeoutTimer: TON:=(PT:=T#120S);
END_VAR

                    _TimeoutTimer(IN:=_Step > 0);
IF _TimeoutTimer.Q THEN
	_Step := 0;
	_Error := TRUE;
	_ErrorDescription := 'timed out waiting for response.';
END_IF

_ResetRtrig(CLK:=_Reset);
IF _ResetRtrig.Q THEN
	_Reset := FALSE;
	_Step := 0;
END_IF

_Done := _Step = 0;
_Busy := NOT _Done;

CASE _Step OF
	0: // IDLE
		IF _Execute THEN
			_Execute := FALSE;
			IF _TcpClient._M_Write(Data:=_Command) THEN
				_ReadRecordLast := _TcpClient.dRecordRead;
				_Step := _Step + 1;
			ELSE
				_Step := 0;
			END_IF
		END_IF
	
	1: // WAIT
		IF _TcpClient.dRecordRead <> _ReadRecordLast THEN
			_ReadRecordLast := _TcpClient.dRecordRead;
			IF find(_TcpClient.strRead, 'res: ') = 1 THEN
				MemUtils.MemSet(
					pbyBuffer:=ADR(_Response),
					byValue:=0,
					dwSize:=SIZEOF(_Response));
				_Response := _TcpClient.strRead;
				_Step := 0;
				
			ELSIF find(_TcpClient.strRead, 'worker uid: ') = 1 THEN
				MemUtils.MemSet(
					pbyBuffer:=ADR(_WorkerUid),
					byValue:=0,
					dwSize:=SIZEOF(_WorkerUid));
				_WorkerUid := DELETE(STR:=_TcpClient.strRead, LEN:=12, POS:=1);
				
			ELSIF find(_TcpClient.strRead, 'command uid: ') = 1 THEN
				MemUtils.MemSet(
					pbyBuffer:=ADR(_WorkerUid),
					byValue:=0,
					dwSize:=SIZEOF(_WorkerUid));
				_WorkerUid := DELETE(STR:=_TcpClient.strRead, LEN:=12, POS:=1);
				
			END_IF
		END_IF
		
END_CASE

_TcpClient(
	bEnable:= TRUE, 
	strIpAddress:= sIpAddress, 
	uPort:= uPort,
	bBusyWrite=> , 
	bDoneWrite=> , 
	bBusyRead=> , 
	dRecordRead=> , 
	strRead=> );
                  

METHOD PROTECTED _M_Execute : BOOL
VAR_INPUT
	Command: STRING(255):='';
	Timeout: UDINT:=60;
END_VAR
                          _Execute := TRUE;
_Command:=Command;
_TimeoutTimer.PT := UDINT_TO_TIME(Timeout * 1000);
                        
END_METHOD

METHOD PUBLIC M_Cancel : BOOL
VAR_INPUT
END_VAR
                          IF _WorkerUid <> '' THEN
	M_Cancel := TRUE;
	_Command := 'kill: ';
	_Command := CONCAT(_Command, _WorkerUid);
	_WorkerUid := ''; // lets make sure to forget this uid in case its used again for something else
	_Step := 0;
	_Execute := TRUE;
	
ELSE
	M_Cancel := FALSE;
	
END_IF
                        
END_METHOD

METHOD PUBLIC M_Reset : BOOL
VAR_INPUT
END_VAR
                          _Reset := TRUE;
_Error := FALSE;
_ErrorDescription := '';
                        
END_METHOD

METHOD PUBLIC M_Reconnect : BOOL
VAR_INPUT
END_VAR
                          _TcpClient._M_Reconnect();
                        
END_METHOD

{attribute 'monitoring':='variable'}
PROPERTY PUBLIC P_Done : BOOL
GET
VAR
END_VAR
                            P_Done := _Done;
                          
END_GET
END_PROPERTY

{attribute 'monitoring':='variable'}
PROPERTY PUBLIC P_Busy : BOOL
GET
VAR
END_VAR
                            P_Busy := _Busy;
                          
END_GET
END_PROPERTY

{attribute 'monitoring':='variable'}
PROPERTY PUBLIC P_Error : BOOL
GET
VAR
END_VAR
                            P_Error := _Error;
                          
END_GET
END_PROPERTY

{attribute 'monitoring':='variable'}
PROPERTY PUBLIC P_ErrorDescription : STRING
GET
VAR
END_VAR
                            P_ErrorDescription := _ErrorDescription;
                          
END_GET
END_PROPERTY

{attribute 'monitoring':='variable'}
PROPERTY PUBLIC P_Response : STRING(255)
GET
VAR
END_VAR
                            P_Response := _Response;
                          
END_GET
END_PROPERTY

{attribute 'monitoring':='variable'}
PROPERTY PUBLIC P_RawReadString : REFERENCE TO STRING(255)
GET
VAR
END_VAR
                            P_RawReadString REF= _TcpClient.strRead;
                          
END_GET
END_PROPERTY

{attribute 'monitoring':='variable'}
PROPERTY PUBLIC P_RawReadByteArray : ARRAY[0..254] OF BYTE
GET
VAR
END_VAR
                            P_RawReadByteArray := _TcpClient.byteArrayRead;
                          
END_GET
END_PROPERTY

{attribute 'monitoring':='variable'}
PROPERTY PUBLIC P_RecordNumber : DINT
GET
VAR
END_VAR
                            P_RecordNumber := _TcpClient.dRecordRead;
                          
END_GET
END_PROPERTY

{attribute 'monitoring':='variable'}
PROPERTY PUBLIC P_Connected : REFERENCE TO BOOL
GET
VAR
END_VAR
                            P_Connected REF= _TcpClient.bConnected;
                          
END_GET
END_PROPERTY
END_FUNCTION_BLOCK

FUNCTION F_DpadState : ST_Dpad
VAR_INPUT
	State: USINT;
END_VAR
VAR
END_VAR

                    CASE State OF
	0:
		F_DpadState.Up := TRUE;
		F_DpadState.Down := FALSE;
		F_DpadState.Left := FALSE;
		F_DpadState.Right := FALSE;
	1:
		F_DpadState.Up := TRUE;
		F_DpadState.Down := FALSE;
		F_DpadState.Left := FALSE;
		F_DpadState.Right := TRUE;
	2:
		F_DpadState.Up := FALSE;
		F_DpadState.Down := FALSE;
		F_DpadState.Left := FALSE;
		F_DpadState.Right := TRUE;
	3:
		F_DpadState.Up := FALSE;
		F_DpadState.Down := TRUE;
		F_DpadState.Left := FALSE;
		F_DpadState.Right := TRUE;
	4:
		F_DpadState.Up := FALSE;
		F_DpadState.Down := TRUE;
		F_DpadState.Left := FALSE;
		F_DpadState.Right := FALSE;
	5:
		F_DpadState.Up := FALSE;
		F_DpadState.Down := TRUE;
		F_DpadState.Left := TRUE;
		F_DpadState.Right := FALSE;
	6:
		F_DpadState.Up := FALSE;
		F_DpadState.Down := FALSE;
		F_DpadState.Left := TRUE;
		F_DpadState.Right := FALSE;
	7:
		F_DpadState.Up := TRUE;
		F_DpadState.Down := FALSE;
		F_DpadState.Left := TRUE;
		F_DpadState.Right := FALSE;
		
ELSE
	F_DpadState.Up := FALSE;
	F_DpadState.Down := FALSE;
	F_DpadState.Left := FALSE;
	F_DpadState.Right := FALSE;
		
END_CASE
                  
END_FUNCTION

FUNCTION_BLOCK FB_GroupHandler
VAR_IN_OUT
	AxisGroup: AXIS_GROUP_REF_SM3;
END_VAR
VAR_INPUT
	Enable: BOOL;
	StoredPositions: REFERENCE TO ARRAY[GVL.POS_ARR_BEG..GVL.POS_ARR_END] OF DUT_StoredPosition;
END_VAR
VAR_OUTPUT
	Busy: BOOL;
	Error: BOOL;
	ErrorID: SMC_ERROR;
END_VAR
VAR
	//
	EnableFtrig: F_TRIG;
	
	//
	_SeqEnableGroup: INT;
	_SeqDisableGroup: INT;
	_SequenceSetKinematics: INT;
	_SequenceSetCoordTrans: INT;
	_SeqResetGroup: INT;
	
	//
	_SMC_GroupPower: SMC_GroupPower;
	_GroupPower: BOOL;
	_MC_GroupEnable: MC_GroupEnable;
	_MC_GroupDisable: MC_GroupDisable;
	_MC_GroupReset: MC_GroupReset;
	_MC_GroupReadActualPosition: MC_GroupReadActualPosition;
	_SMC_SetKinConfiguration: SMC_SetKinConfiguration;
	
    // coordinate transforms
	_MC_SetCoordinateTransform: MC_SetCoordinateTransform;
	_SMC_GroupSetTool: SMC_GroupSetTool;
	_MC_COORD_REF: MC_COORD_REF;
	_CoordinateSystem: SMC_COORD_SYSTEM:=SMC_COORD_SYSTEM.ACS;
	
	_EnableGroup: BOOL;
	_DisableGroup: BOOL;
	_GroupEnabled: BOOL;
	_ResetGroup: BOOL;
	_SetKinematics: BOOL;
	_SetCoordinates: BOOL;
	_KinematicsSet: BOOL;
	
	_MC_GroupReadStatus: MC_GroupReadStatus;
	_DUT_GroupStatus: DUT_GroupStatus;
	
END_VAR

VAR CONSTANT
	STEP_DONE: 				INT := 1000;
	STEP_IDLE: 				INT := 0000;
	STEP_GROUP_POWER_ON: 	INT := 0022;
	STEP_WAIT_POWER_ON: 	INT := 0024;
	STEP_GROUP_ENABLE: 		INT := 0030;
	STEP_WAIT_ENABLE: 		INT := 0035;
	STEP_READ_POSITION: 	INT := 0040;
	STEP_WAIT_POSITION: 	INT := 0050;
	STEP_SET_KINEMATICS: 	INT := 0060;
	STEP_WAIT_KINEMATICS: 	INT := 0070;
	STEP_SET_COORD_TRANS: 	INT := 0071;
	STEP_WAIT_COORD_TRANS: 	INT := 0072;
	STEP_GROUP_DISABLE: 	INT := 0100;
	STEP_WAIT_DISABLE: 		INT := 0110;
	STEP_GROUP_POWER_OFF: 	INT := 0120;
END_VAR

                    //
Busy := _SeqEnableGroup <> 0
		OR _SeqDisableGroup <> 0
		OR _SequenceSetKinematics <> 0
		OR _SequenceSetCoordTrans <> 0
		OR _SeqResetGroup <> 0;
		
EnableFtrig(CLK:=Enable);
IF EnableFtrig.Q THEN
	M_DisableGroup();
END_IF

//
_M_EnableGroup();
_M_DisableGroup();
_M_SetKinematics();
_M_ResetGroup();

_MC_GroupReadStatus(
	AxisGroup:= AxisGroup, 
	Enable:= Enable, 
	Valid=> _DUT_GroupStatus.Valid, 
	Busy=> _DUT_GroupStatus.Busy, 
	Error=> _DUT_GroupStatus.Error, 
	ErrorID=> _DUT_GroupStatus.ErrorID, 
	GroupMoving=> _DUT_GroupStatus.GroupMoving, 
	GroupHoming=> _DUT_GroupStatus.GroupHoming, 
	GroupErrorStop=> _DUT_GroupStatus.GroupErrorStop, 
	GroupStandby=> _DUT_GroupStatus.GroupStandby, 
	GroupStopping=> _DUT_GroupStatus.GroupStopping, 
	GroupDisabled=> _DUT_GroupStatus.GroupDisabled, 
	TrackingDynamicCS=> _DUT_GroupStatus.TrackingDynamicCS, 
	InSync=> _DUT_GroupStatus.InSync, 
	ActiveMovementId=> _DUT_GroupStatus.ActiveMovementId, 
	FirstReferencedMovementId=> _DUT_GroupStatus.FirstReferencedMovementId, 
	LastAcceptedMovementId=> _DUT_GroupStatus.LastAcceptedMovementId, 
	PositionLag=> _DUT_GroupStatus.PositionLag, 
	OrientationLag=> _DUT_GroupStatus.OrientationLag);

_MC_SetCoordinateTransform(
	AxisGroup:= AxisGroup, 
	Execute:= , 
	CoordTransform:= _MC_COORD_REF, 
	CoordSystem:= , 
	Done=> , 
	Busy=> , 
	Error=> , 
	ErrorID=> );

_SMC_GroupSetTool(
	AxisGroup:= AxisGroup, 
	Execute:= , 
	ToolOffset:= _MC_COORD_REF, 
	Done=> , 
	Error=> , 
	ErrorID=> );

_SMC_GroupPower(
	AxisGroup:= AxisGroup, 
	Enable:= _GroupPower, 
	bRegulatorOn:= _GroupPower, 
	bDriveStart:= _GroupPower, 
	Status=> , 
	Busy=> , 
	Error=> , 
	ErrorID=> );

_MC_GroupEnable(
	AxisGroup:= AxisGroup, 
	Execute:= , 
	CompatibilityOptions:= , 
	Done=> , 
	Busy=> , 
	Error=> , 
	ErrorID=> );
	
_MC_GroupDisable(
	AxisGroup:= AxisGroup, 
	Execute:= , 
	Done=> , 
	Busy=> , 
	Error=> , 
	ErrorID=> );

_MC_GroupReset(
	AxisGroup:= AxisGroup, 
	Execute:= , 
	Done=> , 
	Busy=> , 
	Error=> , 
	ErrorID=> );

_MC_GroupReadActualPosition(
	AxisGroup:= AxisGroup, 
	Enable:= , 
	CoordSystem:= _CoordinateSystem, 
	Valid=> , 
	Busy=> , 
	Error=> , 
	ErrorID=> , 
	Position=> , 
	KinematicConfig=> );
	
_SMC_SetKinConfiguration(
	AxisGroup:= AxisGroup, 
	Execute:= , 
	ConfigData:= _MC_GroupReadActualPosition.KinematicConfig, 
	Done=> , 
	Busy=> , 
	Error=> , 
	ErrorID=> );
                  

METHOD PRIVATE _M_EnableGroup : BOOL
VAR_INPUT
END_VAR
                          
CASE _SeqEnableGroup OF
	0: // IDLE
		IF _EnableGroup THEN
			_EnableGroup := FALSE;
			_GroupEnabled := FALSE;
			_MC_GroupEnable.Execute := FALSE;
			_SeqEnableGroup := _SeqEnableGroup + 1;
		END_IF
		
	1:
		_GroupPower := TRUE;
		_SeqEnableGroup := _SeqEnableGroup + 1;
		
	2:
		// TODO add timeout timer here
		IF _SMC_GroupPower.Error THEN
			Error := TRUE;
			ErrorID := _SMC_GroupPower.ErrorID;
			_SeqEnableGroup := 0;
		ELSIF _SMC_GroupPower.Status THEN
			_SeqEnableGroup := _SeqEnableGroup + 1;
		END_IF
		
	3:
		_MC_GroupEnable.Execute := TRUE;
		_SeqEnableGroup := _SeqEnableGroup + 1;
		
	4:
		// TODO add timeout timer here
		IF NOT _MC_GroupEnable.Busy THEN // this is a hack. we need to figure out is the group is already enabled first
			_GroupEnabled := TRUE;
			//_MC_GroupEnable.Execute := FALSE;
			_SeqEnableGroup := 0;
		END_IF;
END_CASE
                        
END_METHOD

METHOD PRIVATE _M_SetKinematics : BOOL
VAR_INPUT
END_VAR
                          
CASE _SequenceSetKinematics OF
	0: // IDLE
		IF _SetKinematics THEN
			_SetKinematics := FALSE;
			_KinematicsSet := FALSE;
			_MC_GroupReadActualPosition.Enable := FALSE;
			_SMC_SetKinConfiguration.Execute := FALSE;
			_SequenceSetKinematics := _SequenceSetKinematics + 1;
		END_IF
		
	1: // read group position
		_MC_GroupReadActualPosition.Enable := TRUE;
		_SequenceSetKinematics := _SequenceSetKinematics + 1;
		
	2: // wait for group read position
		// TODO add timeout timer here
		IF _MC_GroupReadActualPosition.Error THEN
			Error := TRUE;
			ErrorID := _MC_GroupReadActualPosition.ErrorID;
			_SequenceSetKinematics := 0;
		ELSIF _MC_GroupReadActualPosition.Valid THEN
			_SequenceSetKinematics := _SequenceSetKinematics + 1;
		END_IF
		
	3: // set kinematics
        // orientation convention is always ZYZ for softmotion
        GVL.OriConvention := SMC_ORI_CONVENTION.ZYZ;
        //
		_SMC_SetKinConfiguration.Execute := TRUE;
		_SequenceSetKinematics := _SequenceSetKinematics + 1;
		
	4: // wait for set kinematics
		// TODO add timeout timer here
		IF _SMC_SetKinConfiguration.Error THEN
			Error := TRUE;
			ErrorID := _SMC_SetKinConfiguration.ErrorID;
			_SequenceSetKinematics := 0;
		ELSIF _SMC_SetKinConfiguration.Done THEN
			_SMC_SetKinConfiguration.Execute := FALSE;
			_SequenceSetKinematics := _SequenceSetKinematics + 1;
		END_IF
		
	5:
		_SetCoordinates := TRUE;
		_SequenceSetKinematics := _SequenceSetKinematics + 1;
	
	6:
		// TODO add timeout timer here
		IF _MC_SetCoordinateTransform.Error THEN
			Error := TRUE;
			ErrorID := _MC_SetCoordinateTransform.ErrorID;
			_SequenceSetCoordTrans := 0;
			_SequenceSetKinematics := 0;
		ELSIF _SMC_GroupSetTool.Error THEN
			Error := TRUE;
			ErrorID := _SMC_GroupSetTool.ErrorID;
			_SequenceSetCoordTrans := 0;
			_SequenceSetKinematics := 0;
		ELSIF _SequenceSetCoordTrans <= 0 THEN
			_KinematicsSet := TRUE;
			_SequenceSetKinematics := 0;
		END_IF
		
END_CASE

CASE _SequenceSetCoordTrans OF
	0: //
		IF _SetCoordinates THEN
			_SetCoordinates := FALSE;
			_SMC_GroupSetTool.Execute := FALSE;
			_MC_SetCoordinateTransform.Execute := FALSE;
			_SequenceSetCoordTrans := _SequenceSetCoordTrans + 1;
		END_IF
	
	1: //
		_MC_COORD_REF := StoredPositions[GVL.MCS_POS_IDX].Position; // MCS
		_MC_SetCoordinateTransform.CoordSystem := SMC_COORD_SYSTEM.MCS;
		_MC_SetCoordinateTransform.Execute := TRUE;
		_SequenceSetCoordTrans := _SequenceSetCoordTrans + 1;
		
	2: //
		// TODO add timeout timer here
		IF _MC_SetCoordinateTransform.Error THEN
			(*SUPER^.M_Error(Description:=CONCAT('Move Command Error: ',
										CONCAT(TO_STRING(_MC_SetCoordinateTransform.ErrorID),
										CONCAT(' ', SMC_ErrorString(_MC_SetCoordinateTransform.ErrorID,
													SMC_Language_Type.english)))));*)
			_SequenceSetCoordTrans := 10; // error step so we dont spam errors
			
		ELSIF _MC_SetCoordinateTransform.Done THEN
			_MC_SetCoordinateTransform.Execute := FALSE;
			_SequenceSetCoordTrans := _SequenceSetCoordTrans + 1;
		END_IF
		
	3: //
		_MC_COORD_REF := StoredPositions[GVL.PC1_POS_IDX].Position; // PCS 1
		_MC_SetCoordinateTransform.CoordSystem := SMC_COORD_SYSTEM.PCS_1;
		_MC_SetCoordinateTransform.Execute := TRUE;
		_SequenceSetCoordTrans := _SequenceSetCoordTrans + 1;
		
	4: //
		// TODO add timeout timer here
		IF _MC_SetCoordinateTransform.Error THEN
			(*SUPER^.M_Error(Description:=CONCAT('Move Command Error: ',
										CONCAT(TO_STRING(_MC_SetCoordinateTransform.ErrorID),
										CONCAT(' ', SMC_ErrorString(_MC_SetCoordinateTransform.ErrorID,
													SMC_Language_Type.english)))));*)
			_SequenceSetCoordTrans := 10; // error step so we dont spam errors
			
		ELSIF _MC_SetCoordinateTransform.Done THEN
			_MC_SetCoordinateTransform.Execute := FALSE;
			_SequenceSetCoordTrans := _SequenceSetCoordTrans + 1;
		END_IF
		
	5: //
		_MC_COORD_REF := StoredPositions[GVL.PC2_POS_IDX].Position; // PCS 2
		_MC_SetCoordinateTransform.CoordSystem := SMC_COORD_SYSTEM.PCS_2;
		_MC_SetCoordinateTransform.Execute := TRUE;
		_SequenceSetCoordTrans := _SequenceSetCoordTrans + 1;
		
	6: //
		// TODO add timeout timer here
		IF _MC_SetCoordinateTransform.Error THEN
			(*SUPER^.M_Error(Description:=CONCAT('Move Command Error: ',
										CONCAT(TO_STRING(_MC_SetCoordinateTransform.ErrorID),
										CONCAT(' ', SMC_ErrorString(_MC_SetCoordinateTransform.ErrorID,
													SMC_Language_Type.english)))));*)
			_SequenceSetCoordTrans := 10; // error step so we dont spam errors
			
		ELSIF _MC_SetCoordinateTransform.Done THEN
			_MC_SetCoordinateTransform.Execute := FALSE;
			_SequenceSetCoordTrans := _SequenceSetCoordTrans + 1;
		END_IF
		
	7:  // set tool offset
		_MC_COORD_REF := StoredPositions[GVL.TCP_POS_IDX].Position; // TCP
		_SMC_GroupSetTool.Execute := TRUE;
		_SequenceSetCoordTrans := _SequenceSetCoordTrans + 1;
		
	8: // monitor tool offset
		// TODO add timeout timer here
		IF _SMC_GroupSetTool.Error THEN
			(*SUPER^.M_Error(Description:=CONCAT('Move Command Error: ',
										CONCAT(TO_STRING(_SMC_GroupSetTool.ErrorID),
										CONCAT(' ', SMC_ErrorString(_SMC_GroupSetTool.ErrorID,
													SMC_Language_Type.english)))));*)
			_SequenceSetCoordTrans := 999; // error step so we dont spam errors
			
		ELSIF _SMC_GroupSetTool.Done THEN
			_SMC_GroupSetTool.Execute := FALSE;
			_SequenceSetCoordTrans := 0;
		END_IF

END_CASE
                        
END_METHOD

METHOD PRIVATE _M_DisableGroup : BOOL
VAR_INPUT
END_VAR
                          
CASE _SeqDisableGroup OF
	0: // IDLE
		IF _DisableGroup THEN
			_DisableGroup := FALSE;
			_MC_GroupDisable.Execute := FALSE;
			_MC_GroupEnable.Execute := FALSE;
			_SeqDisableGroup := _SeqDisableGroup + 1;
		END_IF
		
	1:
		_MC_GroupDisable.Execute := TRUE;
		_SeqDisableGroup := _SeqDisableGroup + 1;
		
	2:
		// TODO add timeout timer here
		IF NOT _MC_GroupDisable.Busy THEN // this is a hack. we need to figure out is the group is already disabled first
			_SeqDisableGroup := _SeqDisableGroup + 1;;
		END_IF
		
	3:
		_MC_GroupDisable.Execute := FALSE;
		_GroupEnabled := FALSE;
		_KinematicsSet := FALSE;
		_GroupPower := FALSE;
		_SeqDisableGroup := 0;
		
END_CASE
                        
END_METHOD

METHOD PUBLIC M_EnableGroup : BOOL
VAR_INPUT
END_VAR
                          IF Enable AND NOT Error THEN
	M_EnableGroup := TRUE;
	_EnableGroup := TRUE;
	_GroupEnabled := FALSE;
ELSE
	M_EnableGroup := FALSE;
END_IF
                        
END_METHOD

METHOD PRIVATE _M_ResetGroup : BOOL
VAR_INPUT
END_VAR
                          
CASE _SeqResetGroup OF
	0: // IDLE
		IF _ResetGroup THEN
			_ResetGroup := FALSE;
			//IF Error THEN
				_SeqResetGroup := _SeqResetGroup + 1;
			//END_IF
		END_IF
		
	1:
		Error := FALSE;
		ErrorID := SMC_NO_ERROR;
		_MC_GroupReset.Execute := TRUE;
		_SeqResetGroup := _SeqResetGroup + 1;
	
	2: 
		_MC_GroupReset.Execute := FALSE;
		//
		_SeqEnableGroup := 0;
		_SeqDisableGroup := 0;
		_SequenceSetKinematics := 0;
		_SequenceSetCoordTrans := 0;
		_SeqResetGroup := 0;
	
END_CASE
                        
END_METHOD

METHOD PUBLIC M_DisableGroup : BOOL
VAR_INPUT
END_VAR
                          //IF NOT Error THEN
	M_DisableGroup := TRUE;
	_DisableGroup := TRUE;
//ELSE
	//M_DisableGroup := FALSE;
//END_IF
                        
END_METHOD

METHOD PUBLIC M_SetKinematics : BOOL
VAR_INPUT
	CoordinateSystem: SMC_COORD_SYSTEM;
END_VAR
                          IF _GroupEnabled AND NOT Error THEN
	M_SetKinematics := TRUE;
	_CoordinateSystem := CoordinateSystem;
	_SetKinematics := TRUE;
	_KinematicsSet := FALSE;
ELSE
	M_SetKinematics := FALSE;
END_IF
                        
END_METHOD

METHOD PUBLIC M_ResetGroup : BOOL
VAR_INPUT
END_VAR
                          _ResetGroup := TRUE;
                        
END_METHOD

{attribute 'monitoring' := 'variable'}
PROPERTY PUBLIC P_GroupEnabled : BOOL
GET
VAR
END_VAR
                            P_GroupEnabled := _GroupEnabled;
                          
END_GET
END_PROPERTY

{attribute 'monitoring' := 'variable'}
PROPERTY PUBLIC P_KinematicsSet : BOOL
GET
VAR
END_VAR
                            P_KinematicsSet := _KinematicsSet;
                          
END_GET
END_PROPERTY

{attribute 'monitoring' := 'variable'}
PROPERTY PUBLIC P_GroupStatus : REFERENCE TO DUT_GroupStatus
GET
VAR
END_VAR
                            P_GroupStatus REF= _DUT_GroupStatus;
                          
END_GET
END_PROPERTY
END_FUNCTION_BLOCK

FUNCTION F_SetJogButtons : INT
VAR_INPUT
	CoordinateSystem: SMC_COORD_SYSTEM;
	ABC_as_ACS: BOOL;
END_VAR
VAR
END_VAR

                    CASE CoordinateSystem OF
	SMC_COORD_SYSTEM.ACS:
		F_SetJogButtons := 0;
	SMC_COORD_SYSTEM.MCS:
		IF ABC_as_ACS THEN
			F_SetJogButtons := 2;
		ELSE
			F_SetJogButtons := 1;
		END_IF
	SMC_COORD_SYSTEM.PCS_1:
		IF ABC_as_ACS THEN
			F_SetJogButtons:= 2;
		ELSE
			F_SetJogButtons := 1;
		END_IF
	SMC_COORD_SYSTEM.PCS_2:
		IF ABC_as_ACS THEN
			F_SetJogButtons := 2;
		ELSE
			F_SetJogButtons := 1;
		END_IF
	SMC_COORD_SYSTEM.TCS:
		IF ABC_as_ACS THEN
			F_SetJogButtons := 2;
		ELSE
			F_SetJogButtons := 1;
		END_IF
	SMC_COORD_SYSTEM.WCS:
		IF ABC_as_ACS THEN
			F_SetJogButtons := 2;
		ELSE
			F_SetJogButtons := 1;
		END_IF
	ELSE
		F_SetJogButtons := 0;
		
END_CASE
                  
END_FUNCTION

FUNCTION_BLOCK FB_HomingProcessor
VAR_IN_OUT
	J1, J2, J3, J4, J5, J6: AXIS_REF_SM3;
	AxisGroup: AXIS_GROUP_REF_SM3;
	GroupHandler: FB_GroupHandler;
	Controller: FB_Controller;
END_VAR

VAR_INPUT
	J1_Limit, J2_Limit, J3_Limit, J4_Limit, J5_Limit, J6_Limit: BOOL;
	Enable: BOOL;
	Reset: BOOL;
	StoredPositions: REFERENCE TO ARRAY[GVL.POS_ARR_BEG..GVL.POS_ARR_END] OF DUT_StoredPosition;
	VisionRegisters: REFERENCE TO ARRAY[GVL.VIS_ARR_BEG..GVL.VIS_ARR_END] OF DUT_VisionRegister;
	Flags: REFERENCE TO ARRAY[GVL.FLG_ARR_BEG..GVL.FLG_ARR_END] OF DUT_Flags;
END_VAR
VAR_OUTPUT
	Done: BOOL;
	Busy: BOOL;
	Error: BOOL;
	ErrorID: SMC_ERROR;
END_VAR
VAR
	_ExecuteRtrig: R_TRIG;
	_ExecuteFtrig: F_TRIG;
	_ResetRtrig: R_TRIG;
	_ErrorRtrig: R_TRIG;
	
	_SequenceMain: INT;
	_StartHoming: BOOL;
	
	_SMC_Homing_J1, _SMC_Homing_J2, _SMC_Homing_J3: SMC_Homing;
	_SMC_Homing_J4, _SMC_Homing_J5, _SMC_Homing_J6: SMC_Homing;
	
	_MC_SetPosition_J1, _MC_SetPosition_J2, _MC_SetPosition_J3: MC_SetPosition;
	_MC_SetPosition_J4, _MC_SetPosition_J5, _MC_SetPosition_J6: MC_SetPosition;
	
	_HomingVelocityFast: LREAL:= 15.0;
	_HomingVelocitySlow: LREAL:= 10.0;
	_HomingVelocitySlowSlow: LREAL:= 1.0;
	_HomingAcceleration: LREAL:= 50.0;
	_HomingJerk: LREAL:= 100.0;
	
	_MoveToPose: BOOL;
	_MoveCommand: ST_MoveCmd;
	_MoveCommandProcessor: FB_MoveCmdProcessor;
	
	_i, _j, _k: INT;
	_FirstScan: BOOL:=TRUE;
END_VAR

VAR CONSTANT
	STEP_DONE: 					INT := 9999;
	STEP_IDLE: 					INT := 0000;
	STEP_GROUP_ENABLE: 			INT := 0030;
	STEP_WAIT_ENABLE: 			INT := 0035;
	STEP_FAST_HOME_G1:			INT := 0040;
	STEP_WAIT_FAST_HOME_G1:		INT := 0045;
	STEP_SLOW_HOME_G1:			INT := 0050;
	STEP_WAIT_SLOW_HOME_G1:		INT := 0055;
	
	STEP_FAST_HOME_G2:			INT := 0060;
	STEP_WAIT_FAST_HOME_G2:		INT := 0065;
	STEP_SLOW_HOME_G2:			INT := 0070;
	STEP_WAIT_SLOW_HOME_G2:		INT := 0075;
	
	STEP_FAST_HOME_G3:			INT := 0080;
	STEP_WAIT_FAST_HOME_G3:		INT := 0085;
	STEP_SLOW_HOME_G3:			INT := 0090;
	STEP_WAIT_SLOW_HOME_G3:		INT := 0095;
	
	STEP_MOVE_TO_POSE:			INT := 1000;
	STEP_WAIT_MOVE_TO_POSE:		INT := 1010;
	STEP_WAIT_POSE_DONE:		INT := 1020;
END_VAR

                    // TODO refactor all the code in the FB to use arrays and for loops ... whenever you get bored...

_ExecuteRtrig(CLK:=_StartHoming);
_ExecuteFtrig(CLK:=_StartHoming);
_ResetRtrig(CLK:=Reset);

IF _ExecuteRtrig.Q THEN
    _StartHoming := FALSE;
END_IF

IF _FirstScan THEN
	//
END_IF

CASE _SequenceMain OF
	STEP_DONE: // done
		Busy := FALSE;
		Done := TRUE;
		_MoveCommandProcessor.M_Home();
		_SequenceMain := STEP_IDLE;
		
		_SMC_Homing_J1.bExecute := FALSE;
		_SMC_Homing_J2.bExecute := FALSE;
		_SMC_Homing_J3.bExecute := FALSE;
		_SMC_Homing_J4.bExecute := FALSE;
		_SMC_Homing_J5.bExecute := FALSE;
		_SMC_Homing_J6.bExecute := FALSE;
		
		J1.bSWLimitEnable := TRUE;
		J2.bSWLimitEnable := TRUE;
		J3.bSWLimitEnable := TRUE;
		J4.bSWLimitEnable := TRUE;
		J5.bSWLimitEnable := TRUE;
		J6.bSWLimitEnable := TRUE;
		
	STEP_IDLE: // IDLE
		IF _ExecuteRtrig.Q AND Enable THEN
			Busy := TRUE;
			Done := FALSE;
			_SequenceMain := STEP_GROUP_ENABLE;
			Flags[GVL.HOME_COMPLETE].Value := FALSE;
		END_IF
		
	STEP_GROUP_ENABLE:
		IF GroupHandler.M_EnableGroup() THEN
			_SequenceMain := STEP_WAIT_ENABLE;
		ELSE
			_SequenceMain := STEP_DONE;
			Error := TRUE;
			ErrorID := GroupHandler.ErrorID;
		END_IF
		
	STEP_WAIT_ENABLE:
		// TODO add timeout timer here
		IF GroupHandler.P_GroupEnabled THEN
			_SequenceMain := STEP_FAST_HOME_G1;
		END_IF;
		
	STEP_FAST_HOME_G1:	
		_SMC_Homing_J1.bExecute := SEL(PersistentVars.HomingGroupOne.J1, FALSE, TRUE);
		_SMC_Homing_J2.bExecute := SEL(PersistentVars.HomingGroupOne.J2, FALSE, TRUE);
		_SMC_Homing_J3.bExecute := SEL(PersistentVars.HomingGroupOne.J3, FALSE, TRUE);
		_SMC_Homing_J4.bExecute := SEL(PersistentVars.HomingGroupOne.J4, FALSE, TRUE);
		_SMC_Homing_J5.bExecute := SEL(PersistentVars.HomingGroupOne.J5, FALSE, TRUE);
		_SMC_Homing_J6.bExecute := SEL(PersistentVars.HomingGroupOne.J6, FALSE, TRUE);
		
		_SMC_Homing_J1.bReturnToZero := FALSE;
		_SMC_Homing_J2.bReturnToZero := FALSE;
		_SMC_Homing_J3.bReturnToZero := FALSE;
		_SMC_Homing_J4.bReturnToZero := FALSE;
		_SMC_Homing_J5.bReturnToZero := FALSE;
		_SMC_Homing_J6.bReturnToZero := FALSE;
		
		_SMC_Homing_J1.fVelocitySlow := _HomingVelocitySlow;
		_SMC_Homing_J2.fVelocitySlow := _HomingVelocitySlow;
		_SMC_Homing_J3.fVelocitySlow := _HomingVelocitySlow;
		_SMC_Homing_J4.fVelocitySlow := _HomingVelocitySlow;
		_SMC_Homing_J5.fVelocitySlow := _HomingVelocitySlow;
		_SMC_Homing_J6.fVelocitySlow := _HomingVelocitySlow;
		
		J1.bSWLimitEnable := FALSE;
		J2.bSWLimitEnable := FALSE;
		J3.bSWLimitEnable := FALSE;
		J4.bSWLimitEnable := FALSE;
		J5.bSWLimitEnable := FALSE;
		J6.bSWLimitEnable := FALSE;
		
		_SequenceMain := STEP_WAIT_FAST_HOME_G1;
		
	STEP_WAIT_FAST_HOME_G1: // wait fast home group 1
		IF SEL(PersistentVars.HomingGroupOne.J1, TRUE, _SMC_Homing_J1.bDone)
			AND SEL(PersistentVars.HomingGroupOne.J2, TRUE, _SMC_Homing_J2.bDone)
			AND SEL(PersistentVars.HomingGroupOne.J3, TRUE, _SMC_Homing_J3.bDone) 
			AND SEL(PersistentVars.HomingGroupOne.J4, TRUE, _SMC_Homing_J4.bDone) 
			AND SEL(PersistentVars.HomingGroupOne.J5, TRUE, _SMC_Homing_J5.bDone) 
			AND SEL(PersistentVars.HomingGroupOne.J6, TRUE, _SMC_Homing_J6.bDone) THEN
				_SMC_Homing_J1.bExecute := FALSE;
				_SMC_Homing_J2.bExecute := FALSE;
				_SMC_Homing_J3.bExecute := FALSE;
				_SMC_Homing_J4.bExecute := FALSE;
				_SMC_Homing_J5.bExecute := FALSE;
				_SMC_Homing_J6.bExecute := FALSE;
				
				_SequenceMain := STEP_SLOW_HOME_G1;
		END_IF
		
	STEP_SLOW_HOME_G1: // slow home group 1
		_SMC_Homing_J1.bExecute := SEL(PersistentVars.HomingGroupOne.J1, FALSE, TRUE);
		_SMC_Homing_J2.bExecute := SEL(PersistentVars.HomingGroupOne.J2, FALSE, TRUE);
		_SMC_Homing_J3.bExecute := SEL(PersistentVars.HomingGroupOne.J3, FALSE, TRUE);
		_SMC_Homing_J4.bExecute := SEL(PersistentVars.HomingGroupOne.J4, FALSE, TRUE);
		_SMC_Homing_J5.bExecute := SEL(PersistentVars.HomingGroupOne.J5, FALSE, TRUE);
		_SMC_Homing_J6.bExecute := SEL(PersistentVars.HomingGroupOne.J6, FALSE, TRUE);
		
		_SMC_Homing_J1.bReturnToZero := TRUE;
		_SMC_Homing_J2.bReturnToZero := TRUE;
		_SMC_Homing_J3.bReturnToZero := TRUE;
		_SMC_Homing_J4.bReturnToZero := TRUE;
		_SMC_Homing_J5.bReturnToZero := TRUE;
		_SMC_Homing_J6.bReturnToZero := TRUE;
		
		_SMC_Homing_J1.fVelocitySlow := _HomingVelocitySlowSlow;
		_SMC_Homing_J2.fVelocitySlow := _HomingVelocitySlowSlow;
		_SMC_Homing_J3.fVelocitySlow := _HomingVelocitySlowSlow;
		_SMC_Homing_J4.fVelocitySlow := _HomingVelocitySlowSlow;
		_SMC_Homing_J5.fVelocitySlow := _HomingVelocitySlowSlow;
		_SMC_Homing_J6.fVelocitySlow := _HomingVelocitySlowSlow;
		
		_SequenceMain := STEP_WAIT_SLOW_HOME_G1;
		
	STEP_WAIT_SLOW_HOME_G1:
		IF SEL(PersistentVars.HomingGroupOne.J1, TRUE, _SMC_Homing_J1.bDone)
			AND SEL(PersistentVars.HomingGroupOne.J2, TRUE, _SMC_Homing_J2.bDone)
			AND SEL(PersistentVars.HomingGroupOne.J3, TRUE, _SMC_Homing_J3.bDone) 
			AND SEL(PersistentVars.HomingGroupOne.J4, TRUE, _SMC_Homing_J4.bDone) 
			AND SEL(PersistentVars.HomingGroupOne.J5, TRUE, _SMC_Homing_J5.bDone) 
			AND SEL(PersistentVars.HomingGroupOne.J6, TRUE, _SMC_Homing_J6.bDone) THEN
				_SMC_Homing_J1.bExecute := FALSE;
				_SMC_Homing_J2.bExecute := FALSE;
				_SMC_Homing_J3.bExecute := FALSE;
				_SMC_Homing_J4.bExecute := FALSE;
				_SMC_Homing_J5.bExecute := FALSE;
				_SMC_Homing_J6.bExecute := FALSE;
				
				_SequenceMain := STEP_FAST_HOME_G2;
		END_IF
		
	STEP_FAST_HOME_G2:
		_SMC_Homing_J1.bExecute := SEL(PersistentVars.HomingGroupTwo.J1, FALSE, TRUE);
		_SMC_Homing_J2.bExecute := SEL(PersistentVars.HomingGroupTwo.J2, FALSE, TRUE);
		_SMC_Homing_J3.bExecute := SEL(PersistentVars.HomingGroupTwo.J3, FALSE, TRUE);
		_SMC_Homing_J4.bExecute := SEL(PersistentVars.HomingGroupTwo.J4, FALSE, TRUE);
		_SMC_Homing_J5.bExecute := SEL(PersistentVars.HomingGroupTwo.J5, FALSE, TRUE);
		_SMC_Homing_J6.bExecute := SEL(PersistentVars.HomingGroupTwo.J6, FALSE, TRUE);
		
		_SMC_Homing_J1.bReturnToZero := FALSE;
		_SMC_Homing_J2.bReturnToZero := FALSE;
		_SMC_Homing_J3.bReturnToZero := FALSE;
		_SMC_Homing_J4.bReturnToZero := FALSE;
		_SMC_Homing_J5.bReturnToZero := FALSE;
		_SMC_Homing_J6.bReturnToZero := FALSE;
		
		_SMC_Homing_J1.fVelocitySlow := _HomingVelocitySlow;
		_SMC_Homing_J2.fVelocitySlow := _HomingVelocitySlow;
		_SMC_Homing_J3.fVelocitySlow := _HomingVelocitySlow;
		_SMC_Homing_J4.fVelocitySlow := _HomingVelocitySlow;
		_SMC_Homing_J5.fVelocitySlow := _HomingVelocitySlow;
		_SMC_Homing_J6.fVelocitySlow := _HomingVelocitySlow;

		_SequenceMain := STEP_WAIT_FAST_HOME_G2;
		
	STEP_WAIT_FAST_HOME_G2:
		IF SEL(PersistentVars.HomingGroupTwo.J1, TRUE, _SMC_Homing_J1.bDone)
			AND SEL(PersistentVars.HomingGroupTwo.J2, TRUE, _SMC_Homing_J2.bDone)
			AND SEL(PersistentVars.HomingGroupTwo.J3, TRUE, _SMC_Homing_J3.bDone) 
			AND SEL(PersistentVars.HomingGroupTwo.J4, TRUE, _SMC_Homing_J4.bDone) 
			AND SEL(PersistentVars.HomingGroupTwo.J5, TRUE, _SMC_Homing_J5.bDone) 
			AND SEL(PersistentVars.HomingGroupTwo.J6, TRUE, _SMC_Homing_J6.bDone) THEN
				_SMC_Homing_J1.bExecute := FALSE;
				_SMC_Homing_J2.bExecute := FALSE;
				_SMC_Homing_J3.bExecute := FALSE;
				_SMC_Homing_J4.bExecute := FALSE;
				_SMC_Homing_J5.bExecute := FALSE;
				_SMC_Homing_J6.bExecute := FALSE;
				
				_SequenceMain := STEP_SLOW_HOME_G2;
		END_IF
		
	STEP_SLOW_HOME_G2:
		_SMC_Homing_J1.bExecute := SEL(PersistentVars.HomingGroupTwo.J1, FALSE, TRUE);
		_SMC_Homing_J2.bExecute := SEL(PersistentVars.HomingGroupTwo.J2, FALSE, TRUE);
		_SMC_Homing_J3.bExecute := SEL(PersistentVars.HomingGroupTwo.J3, FALSE, TRUE);
		_SMC_Homing_J4.bExecute := SEL(PersistentVars.HomingGroupTwo.J4, FALSE, TRUE);
		_SMC_Homing_J5.bExecute := SEL(PersistentVars.HomingGroupTwo.J5, FALSE, TRUE);
		_SMC_Homing_J6.bExecute := SEL(PersistentVars.HomingGroupTwo.J6, FALSE, TRUE);
		
		_SMC_Homing_J1.bReturnToZero := TRUE;
		_SMC_Homing_J2.bReturnToZero := TRUE;
		_SMC_Homing_J3.bReturnToZero := TRUE;
		_SMC_Homing_J4.bReturnToZero := TRUE;
		_SMC_Homing_J5.bReturnToZero := TRUE;
		_SMC_Homing_J6.bReturnToZero := TRUE;
		
		_SMC_Homing_J1.fVelocitySlow := _HomingVelocitySlowSlow;
		_SMC_Homing_J2.fVelocitySlow := _HomingVelocitySlowSlow;
		_SMC_Homing_J3.fVelocitySlow := _HomingVelocitySlowSlow;
		_SMC_Homing_J4.fVelocitySlow := _HomingVelocitySlowSlow;
		_SMC_Homing_J5.fVelocitySlow := _HomingVelocitySlowSlow;
		_SMC_Homing_J6.fVelocitySlow := _HomingVelocitySlowSlow;
		
		_SequenceMain := STEP_WAIT_SLOW_HOME_G2;
		
	STEP_WAIT_SLOW_HOME_G2:
		IF SEL(PersistentVars.HomingGroupTwo.J1, TRUE, _SMC_Homing_J1.bDone)
			AND SEL(PersistentVars.HomingGroupTwo.J2, TRUE, _SMC_Homing_J2.bDone)
			AND SEL(PersistentVars.HomingGroupTwo.J3, TRUE, _SMC_Homing_J3.bDone) 
			AND SEL(PersistentVars.HomingGroupTwo.J4, TRUE, _SMC_Homing_J4.bDone) 
			AND SEL(PersistentVars.HomingGroupTwo.J5, TRUE, _SMC_Homing_J5.bDone) 
			AND SEL(PersistentVars.HomingGroupTwo.J6, TRUE, _SMC_Homing_J6.bDone) THEN
				_SMC_Homing_J1.bExecute := FALSE;
				_SMC_Homing_J2.bExecute := FALSE;
				_SMC_Homing_J3.bExecute := FALSE;
				_SMC_Homing_J4.bExecute := FALSE;
				_SMC_Homing_J5.bExecute := FALSE;
				_SMC_Homing_J6.bExecute := FALSE;
				
				_SequenceMain := STEP_FAST_HOME_G3;
		END_IF
		
	STEP_FAST_HOME_G3:
		_SMC_Homing_J1.bExecute := SEL(PersistentVars.HomingGroupThree.J1, FALSE, TRUE);
		_SMC_Homing_J2.bExecute := SEL(PersistentVars.HomingGroupThree.J2, FALSE, TRUE);
		_SMC_Homing_J3.bExecute := SEL(PersistentVars.HomingGroupThree.J3, FALSE, TRUE);
		_SMC_Homing_J4.bExecute := SEL(PersistentVars.HomingGroupThree.J4, FALSE, TRUE);
		_SMC_Homing_J5.bExecute := SEL(PersistentVars.HomingGroupThree.J5, FALSE, TRUE);
		_SMC_Homing_J6.bExecute := SEL(PersistentVars.HomingGroupThree.J6, FALSE, TRUE);
		
		_SMC_Homing_J1.bReturnToZero := FALSE;
		_SMC_Homing_J2.bReturnToZero := FALSE;
		_SMC_Homing_J3.bReturnToZero := FALSE;
		_SMC_Homing_J4.bReturnToZero := FALSE;
		_SMC_Homing_J5.bReturnToZero := FALSE;
		_SMC_Homing_J6.bReturnToZero := FALSE;
		
		_SMC_Homing_J1.fVelocitySlow := _HomingVelocitySlow;
		_SMC_Homing_J2.fVelocitySlow := _HomingVelocitySlow;
		_SMC_Homing_J3.fVelocitySlow := _HomingVelocitySlow;
		_SMC_Homing_J4.fVelocitySlow := _HomingVelocitySlow;
		_SMC_Homing_J5.fVelocitySlow := _HomingVelocitySlow;
		_SMC_Homing_J6.fVelocitySlow := _HomingVelocitySlow;
		
		_SequenceMain := STEP_WAIT_FAST_HOME_G3;
		
	STEP_WAIT_FAST_HOME_G3:
		IF SEL(PersistentVars.HomingGroupThree.J1, TRUE, _SMC_Homing_J1.bDone)
			AND SEL(PersistentVars.HomingGroupThree.J2, TRUE, _SMC_Homing_J2.bDone)
			AND SEL(PersistentVars.HomingGroupThree.J3, TRUE, _SMC_Homing_J3.bDone) 
			AND SEL(PersistentVars.HomingGroupThree.J4, TRUE, _SMC_Homing_J4.bDone) 
			AND SEL(PersistentVars.HomingGroupThree.J5, TRUE, _SMC_Homing_J5.bDone) 
			AND SEL(PersistentVars.HomingGroupThree.J6, TRUE, _SMC_Homing_J6.bDone) THEN
				_SMC_Homing_J1.bExecute := FALSE;
				_SMC_Homing_J2.bExecute := FALSE;
				_SMC_Homing_J3.bExecute := FALSE;
				_SMC_Homing_J4.bExecute := FALSE;
				_SMC_Homing_J5.bExecute := FALSE;
				_SMC_Homing_J6.bExecute := FALSE;
				
				_SequenceMain := STEP_SLOW_HOME_G3;
		END_IF
		
	STEP_SLOW_HOME_G3:
		_SMC_Homing_J1.bExecute := SEL(PersistentVars.HomingGroupThree.J1, FALSE, TRUE);
		_SMC_Homing_J2.bExecute := SEL(PersistentVars.HomingGroupThree.J2, FALSE, TRUE);
		_SMC_Homing_J3.bExecute := SEL(PersistentVars.HomingGroupThree.J3, FALSE, TRUE);
		_SMC_Homing_J4.bExecute := SEL(PersistentVars.HomingGroupThree.J4, FALSE, TRUE);
		_SMC_Homing_J5.bExecute := SEL(PersistentVars.HomingGroupThree.J5, FALSE, TRUE);
		_SMC_Homing_J6.bExecute := SEL(PersistentVars.HomingGroupThree.J6, FALSE, TRUE);
		
		_SMC_Homing_J1.bReturnToZero := TRUE;
		_SMC_Homing_J2.bReturnToZero := TRUE;
		_SMC_Homing_J3.bReturnToZero := TRUE;
		_SMC_Homing_J4.bReturnToZero := TRUE;
		_SMC_Homing_J5.bReturnToZero := TRUE;
		_SMC_Homing_J6.bReturnToZero := TRUE;
		
		_SMC_Homing_J1.fVelocitySlow := _HomingVelocitySlowSlow;
		_SMC_Homing_J2.fVelocitySlow := _HomingVelocitySlowSlow;
		_SMC_Homing_J3.fVelocitySlow := _HomingVelocitySlowSlow;
		_SMC_Homing_J4.fVelocitySlow := _HomingVelocitySlowSlow;
		_SMC_Homing_J5.fVelocitySlow := _HomingVelocitySlowSlow;
		_SMC_Homing_J6.fVelocitySlow := _HomingVelocitySlowSlow;
		
		_SequenceMain := STEP_WAIT_SLOW_HOME_G3;
		
	STEP_WAIT_SLOW_HOME_G3:
		IF SEL(PersistentVars.HomingGroupThree.J1, TRUE, _SMC_Homing_J1.bDone)
			AND SEL(PersistentVars.HomingGroupThree.J2, TRUE, _SMC_Homing_J2.bDone)
			AND SEL(PersistentVars.HomingGroupThree.J3, TRUE, _SMC_Homing_J3.bDone) 
			AND SEL(PersistentVars.HomingGroupThree.J4, TRUE, _SMC_Homing_J4.bDone) 
			AND SEL(PersistentVars.HomingGroupThree.J5, TRUE, _SMC_Homing_J5.bDone) 
			AND SEL(PersistentVars.HomingGroupThree.J6, TRUE, _SMC_Homing_J6.bDone) THEN
				_SMC_Homing_J1.bExecute := FALSE;
				_SMC_Homing_J2.bExecute := FALSE;
				_SMC_Homing_J3.bExecute := FALSE;
				_SMC_Homing_J4.bExecute := FALSE;
				_SMC_Homing_J5.bExecute := FALSE;
				_SMC_Homing_J6.bExecute := FALSE;
				
				Flags[GVL.HOME_COMPLETE].Value := TRUE;
				IF NOT Flags[GVL.HOM_TO_POSE_IDX].Value THEN
					_SequenceMain := STEP_DONE;
				ELSE
					_SequenceMain := STEP_MOVE_TO_POSE;
				END_IF
		END_IF;
		
	STEP_MOVE_TO_POSE:
		_MoveToPose := TRUE;
		_SequenceMain := STEP_WAIT_MOVE_TO_POSE;
	
	STEP_WAIT_MOVE_TO_POSE:
		IF _MoveCommandProcessor.ItfUnitMode.CurrentState <> PACK_ML.State.Idle THEN
			_SequenceMain := STEP_WAIT_POSE_DONE;
		END_IF
		
	STEP_WAIT_POSE_DONE:
		IF _MoveCommandProcessor.ItfUnitMode.CurrentState = PACK_ML.State.Idle THEN
			_SequenceMain := STEP_DONE;
		END_IF
	
END_CASE

_M_HandlePose(AxisGroup:=AxisGroup, GroupHandler:=GroupHandler);

//
IF _ResetRtrig.Q AND Error THEN
	Error := FALSE;
	ErrorID := SMC_NO_ERROR;
	_SequenceMain := STEP_DONE;
	GroupHandler.M_ResetGroup();
	_MoveCommandProcessor.M_Home();
END_IF

//
_ErrorRtrig(CLK:=GroupHandler.Error
				OR _SMC_Homing_J1.bError
				OR _SMC_Homing_J2.bError
				OR _SMC_Homing_J3.bError
				OR _SMC_Homing_J4.bError
				OR _SMC_Homing_J5.bError
				OR _SMC_Homing_J6.bError
				OR _MoveCommandProcessor.Error);			
IF _ErrorRtrig.Q THEN
	Error := TRUE;
	IF GroupHandler.Error THEN
		ErrorID := GroupHandler.ErrorID;
	ELSIF _SMC_Homing_J1.bError THEN
		ErrorID := _SMC_Homing_J1.nErrorID;
	ELSIF _SMC_Homing_J2.bError THEN
		ErrorID := _SMC_Homing_J2.nErrorID;
	ELSIF _SMC_Homing_J3.bError THEN
		ErrorID := _SMC_Homing_J3.nErrorID;
	ELSIF _SMC_Homing_J4.bError THEN
		ErrorID := _SMC_Homing_J4.nErrorID;
	ELSIF _SMC_Homing_J5.bError THEN
		ErrorID := _SMC_Homing_J5.nErrorID;
	ELSIF _SMC_Homing_J6.bError THEN
		ErrorID := _SMC_Homing_J6.nErrorID;
	ELSIF _MoveCommandProcessor.Error THEN
		// TODO need to rework how error messages are handled (globally)
		// if the move command processor has an error, we dont know what it is.
	END_IF
END_IF

// TODO make search direction configurable for any robot
//
_SMC_Homing_J1(
	Axis:=J1 , 
	bExecute:= ,
	fHomePosition:= StoredPositions[GVL.HOM_POS_IDX].Position.X, 
	fVelocitySlow:= , 
	fVelocityFast:= _HomingVelocityFast, 
	fAcceleration:= _HomingAcceleration, 
	fDeceleration:= _HomingAcceleration, 
	fJerk:= _HomingJerk, 
	nDirection:= MC_direction.negative, 
	bReferenceSwitch:= NOT J1_Limit, 
	fSignalDelay:= , 
	nHomingMode:= , 
	bReturnToZero:= , 
	bIndexOccured:= , 
	fIndexPosition:= , 
	bIgnoreHWLimit:= TRUE, 
	bDone=> , 
	bBusy=> , 
	bCommandAborted=> , 
	bError=> , 
	nErrorID=> , 
	bStartLatchingIndex=> );
	
_SMC_Homing_J2(
	Axis:=J2 , 
	bExecute:= , 
	fHomePosition:= StoredPositions[GVL.HOM_POS_IDX].Position.Y,  
	fVelocitySlow:= , 
	fVelocityFast:= _HomingVelocityFast, 
	fAcceleration:= _HomingAcceleration, 
	fDeceleration:= _HomingAcceleration,
	fJerk:= _HomingJerk, 
	nDirection:= MC_Direction.negative, 
	bReferenceSwitch:= NOT J2_Limit, 
	fSignalDelay:= , 
	nHomingMode:= , 
	bReturnToZero:= , 
	bIndexOccured:= , 
	fIndexPosition:= , 
	bIgnoreHWLimit:= TRUE, 
	bDone=> , 
	bBusy=> , 
	bCommandAborted=> , 
	bError=> , 
	nErrorID=> , 
	bStartLatchingIndex=> );
	
_SMC_Homing_J3(
	Axis:=J3 , 
	bExecute:= , 
	fHomePosition:= StoredPositions[GVL.HOM_POS_IDX].Position.Z, 
	fVelocitySlow:= , 
	fVelocityFast:= _HomingVelocityFast, 
	fAcceleration:= _HomingAcceleration, 
	fDeceleration:= _HomingAcceleration,
	fJerk:= _HomingJerk, 
	nDirection:= MC_Direction.positive, 
	bReferenceSwitch:= NOT J3_Limit, 
	fSignalDelay:= , 
	nHomingMode:= , 
	bReturnToZero:= , 
	bIndexOccured:= , 
	fIndexPosition:= , 
	bIgnoreHWLimit:= TRUE, 
	bDone=> , 
	bBusy=> , 
	bCommandAborted=> , 
	bError=> , 
	nErrorID=> , 
	bStartLatchingIndex=> );
	
_SMC_Homing_J4(
	Axis:=J4 , 
	bExecute:= ,
	fHomePosition:= StoredPositions[GVL.HOM_POS_IDX].Position.A, 
	fVelocitySlow:= , 
	fVelocityFast:= _HomingVelocityFast, 
	fAcceleration:= _HomingAcceleration, 
	fDeceleration:= _HomingAcceleration,
	fJerk:= _HomingJerk, 
	nDirection:= MC_Direction.positive, 
	bReferenceSwitch:= NOT J4_Limit, 
	fSignalDelay:= , 
	nHomingMode:= , 
	bReturnToZero:= , 
	bIndexOccured:= , 
	fIndexPosition:= , 
	bIgnoreHWLimit:= TRUE, 
	bDone=> , 
	bBusy=> , 
	bCommandAborted=> , 
	bError=> , 
	nErrorID=> , 
	bStartLatchingIndex=> );
	
_SMC_Homing_J5(
	Axis:=J5 , 
	bExecute:= , 
	fHomePosition:= StoredPositions[GVL.HOM_POS_IDX].Position.B,  
	fVelocitySlow:= , 
	fVelocityFast:= _HomingVelocityFast, 
	fAcceleration:= _HomingAcceleration, 
	fDeceleration:= _HomingAcceleration,
	fJerk:= _HomingJerk, 
	nDirection:= MC_Direction.positive, 
	bReferenceSwitch:= NOT J5_Limit, 
	fSignalDelay:= , 
	nHomingMode:= , 
	bReturnToZero:= , 
	bIndexOccured:= , 
	fIndexPosition:= , 
	bIgnoreHWLimit:= TRUE, 
	bDone=> , 
	bBusy=> , 
	bCommandAborted=> , 
	bError=> , 
	nErrorID=> , 
	bStartLatchingIndex=> );
	
_SMC_Homing_J6(
	Axis:=J6 , 
	bExecute:= , 
	fHomePosition:= StoredPositions[GVL.HOM_POS_IDX].Position.C, 
	fVelocitySlow:= , 
	fVelocityFast:= _HomingVelocityFast, 
	fAcceleration:= _HomingAcceleration, 
	fDeceleration:= _HomingAcceleration,
	fJerk:= _HomingJerk, 
	nDirection:= MC_Direction.negative, 
	bReferenceSwitch:= NOT J6_Limit, 
	fSignalDelay:= , 
	nHomingMode:= , 
	bReturnToZero:= , 
	bIndexOccured:= , 
	fIndexPosition:= , 
	bIgnoreHWLimit:= TRUE, 
	bDone=> , 
	bBusy=> , 
	bCommandAborted=> , 
	bError=> , 
	nErrorID=> , 
	bStartLatchingIndex=> );
	
//
_MC_SetPosition_J1(
	Axis:= J1, 
	Execute:= _MC_SetPosition_J1.Execute AND NOT _MC_SetPosition_J1.Done AND NOT _MC_SetPosition_J1.Error, 
	Position:= 0.0, 
	Mode:= FALSE, // true=relative false=absolute
	Done=> , 
	Busy=> , 
	Error=> , 
	ErrorID=> );
_MC_SetPosition_J2(
	Axis:= J2, 
	Execute:= _MC_SetPosition_J2.Execute AND NOT _MC_SetPosition_J2.Done AND NOT _MC_SetPosition_J2.Error, 
	Position:= 0.0, 
	Mode:= FALSE, // true=relative false=absolute
	Done=> , 
	Busy=> , 
	Error=> , 
	ErrorID=> );
_MC_SetPosition_J3(
	Axis:= J3, 
	Execute:= _MC_SetPosition_J3.Execute AND NOT _MC_SetPosition_J3.Done AND NOT _MC_SetPosition_J3.Error, 
	Position:= 0.0, 
	Mode:= FALSE, // true=relative false=absolute
	Done=> , 
	Busy=> , 
	Error=> , 
	ErrorID=> );
_MC_SetPosition_J4(
	Axis:= J4, 
	Execute:= _MC_SetPosition_J4.Execute AND NOT _MC_SetPosition_J4.Done AND NOT _MC_SetPosition_J4.Error, 
	Position:= 0.0, 
	Mode:= FALSE, // true=relative false=absolute
	Done=> , 
	Busy=> , 
	Error=> , 
	ErrorID=> );
_MC_SetPosition_J5(
	Axis:= J5, 
	Execute:= _MC_SetPosition_J5.Execute AND NOT _MC_SetPosition_J5.Done AND NOT _MC_SetPosition_J5.Error, 
	Position:= 0.0, 
	Mode:= FALSE, // true=relative false=absolute
	Done=> , 
	Busy=> , 
	Error=> , 
	ErrorID=> );
_MC_SetPosition_J6(
	Axis:= J6, 
	Execute:= _MC_SetPosition_J6.Execute AND NOT _MC_SetPosition_J6.Done AND NOT _MC_SetPosition_J6.Error, 
	Position:= 0.0, 
	Mode:= FALSE, // true=relative false=absolute
	Done=> , 
	Busy=> , 
	Error=> , 
	ErrorID=> );
                  

METHOD PUBLIC M_SetHome : BOOL
VAR_INPUT
END_VAR
                          {warning disable C0371}
// adjust all the persistent variables to take on the calibrated values
StoredPositions[GVL.HOM_POS_IDX].Position.X := F_HomeOffsetCalc(	CurrentOffset:= PersistentVars.StoredPositions[GVL.HOM_POS_IDX].Position.X, 
																				CurrentPosition:= J1.fActPosition, 
																				HomeSearchDirection:= _SMC_Homing_J1.nDirection);

StoredPositions[GVL.HOM_POS_IDX].Position.Y := F_HomeOffsetCalc(	CurrentOffset:= PersistentVars.StoredPositions[GVL.HOM_POS_IDX].Position.Y, 
																				CurrentPosition:= J2.fActPosition, 
																				HomeSearchDirection:= _SMC_Homing_J2.nDirection);

StoredPositions[GVL.HOM_POS_IDX].Position.Z := F_HomeOffsetCalc(	CurrentOffset:= PersistentVars.StoredPositions[GVL.HOM_POS_IDX].Position.Z, 
																				CurrentPosition:= J3.fActPosition, 
																				HomeSearchDirection:= _SMC_Homing_J3.nDirection);

StoredPositions[GVL.HOM_POS_IDX].Position.A := F_HomeOffsetCalc(	CurrentOffset:= PersistentVars.StoredPositions[GVL.HOM_POS_IDX].Position.A, 
																				CurrentPosition:= J4.fActPosition, 
																				HomeSearchDirection:= _SMC_Homing_J4.nDirection);

StoredPositions[GVL.HOM_POS_IDX].Position.B := F_HomeOffsetCalc(	CurrentOffset:= PersistentVars.StoredPositions[GVL.HOM_POS_IDX].Position.B, 
																				CurrentPosition:= J5.fActPosition, 
																				HomeSearchDirection:= _SMC_Homing_J5.nDirection);

StoredPositions[GVL.HOM_POS_IDX].Position.C := F_HomeOffsetCalc(	CurrentOffset:= PersistentVars.StoredPositions[GVL.HOM_POS_IDX].Position.C, 
																				CurrentPosition:= J6.fActPosition, 
																				HomeSearchDirection:= _SMC_Homing_J6.nDirection);

// this isnt totally needed but will calibrate the current session without the need to rehome
_MC_SetPosition_J1.Execute:=TRUE;
_MC_SetPosition_J2.Execute:=TRUE;
_MC_SetPosition_J3.Execute:=TRUE;
_MC_SetPosition_J4.Execute:=TRUE;
_MC_SetPosition_J5.Execute:=TRUE;
_MC_SetPosition_J6.Execute:=TRUE;
{warning restore C0371}
                        
END_METHOD

METHOD PUBLIC M_StartHoming : BOOL
VAR_INPUT
END_VAR
                          IF _SequenceMain = STEP_IDLE THEN
	M_StartHoming := TRUE;
	_StartHoming := TRUE;
ELSE
	M_StartHoming := FALSE;
END_IF
                        
END_METHOD

METHOD PRIVATE _M_HandlePose : BOOL
VAR_IN_OUT
	AxisGroup: AXIS_GROUP_REF_SM3;
	GroupHandler: FB_GroupHandler;
END_VAR
VAR_INPUT
END_VAR
VAR
	_MoveCommand: ST_MoveCmd;
	_PoseSpeed: LREAL:=20.0;
END_VAR
                          IF _MoveToPose THEN
	_MoveToPose:= FALSE;
	//
	IF GVL.Enable 
		AND_THEN Flags[GVL.HOME_COMPLETE].Value
		AND_THEN NOT _MoveCommandProcessor.Busy
		AND_THEN NOT _MoveCommandProcessor.Error THEN
			//
			_MoveCommand.MoveType 			:= DUT_Command_MoveType.DirectMove;
			_MoveCommand.PositionType 		:= DUT_Command_PositionType.AbsolutePosition;
			_MoveCommand.CoordinateType 	:= DUT_Command_CoordinateType.Literal;
			_MoveCommand.Speed 				:= _PoseSpeed;
			_MoveCommand.CoordSystem 		:= SMC_COORD_SYSTEM.ACS;
			_MoveCommand.CoordRef 			:= StoredPositions[GVL.POSE_2_IDX].Position;
			//
			_MoveCommandProcessor.Command := F_BuildMoveCmd(_MoveCommand);
			_MoveCommandProcessor.M_Start();
	END_IF;
END_IF

_MoveCommandProcessor(
	StoredPositions:= StoredPositions,
	VisionRegisters:= VisionRegisters,
	Flags:= Flags,
	AxisGroup:= AxisGroup, 
	GroupHandler:= GroupHandler,
	Velocity:= StoredPositions[GVL.SPEEDS_IDX].Position.X, 
	VelFactor:= StoredPositions[GVL.SPEEDS_IDX].Position.A,
	Acceleration:= StoredPositions[GVL.SPEEDS_IDX].Position.Y, 
	AccFactor:= StoredPositions[GVL.SPEEDS_IDX].Position.B,
	Jerk:= StoredPositions[GVL.SPEEDS_IDX].Position.Z,
	JerkFactor:= StoredPositions[GVL.SPEEDS_IDX].Position.C, 
	Position=> ,
	ItfUnitMode=> , 
	Error=> );
                        
END_METHOD
END_FUNCTION_BLOCK

FUNCTION F_VarSetCmdOperate : LREAL
VAR_INPUT
	Operand1: LREAL;
	Operation: DUT_VarSetCmd_OperType;
	Operand2: LREAL;
END_VAR
VAR
	_epsilon : REAL := 0.00000001;
END_VAR

                    CASE Operation OF
	DUT_VarSetCmd_OperType.NOP:
		F_VarSetCmdOperate := Operand1;
		
	DUT_VarSetCmd_OperType.EQUALS:
		F_VarSetCmdOperate := Operand2;
		
	DUT_VarSetCmd_OperType.PLUS:
		F_VarSetCmdOperate := Operand1 + Operand2;
		
	DUT_VarSetCmd_OperType.MINUS:
		F_VarSetCmdOperate := Operand1 - Operand2;
		
	DUT_VarSetCmd_OperType.TIMES:
		F_VarSetCmdOperate := Operand1 * Operand2;
		
	DUT_VarSetCmd_OperType.DIVIDED_BY:
		IF Operand2 <> 0 THEN
			F_VarSetCmdOperate := Operand1 / Operand2;
		ELSE
			F_VarSetCmdOperate := Operand1 / _epsilon;
		END_IF
		
END_CASE
                  
END_FUNCTION

FUNCTION F_Checksum : UINT
VAR_INPUT
	data: POINTER TO BYTE;
	length: UINT;
END_VAR
VAR
	curr_crc: UINT;
	sum1, sum2: USINT;
	_i, _j, _k: UINT;
END_VAR

                    // https://www.tutorialspoint.com/cyclic-redundancy-check-crc-in-arduino
curr_crc := 16#0000;
sum1 := UINT_TO_USINT(curr_crc);
sum2 := UINT_TO_USINT(SHR(curr_crc, 8));
FOR _i:=0 TO length - 1 BY 1 DO
	sum1 := (sum1 + data[_i]) MOD 255;
	sum2 := (sum2 + sum1) MOD 255;
END_FOR
{warning disable C0308}
F_Checksum := SHL(sum2, 8) OR sum1;
{warning restore C0308}
                  
END_FUNCTION

PROGRAM _50_Retains
VAR
	//
	SaveRetain, RestoreRetain: BOOL;
	pApplication : POINTER TO CmpApp.APPLICATION;
	ResultFind, ResultStore, ResultRestore: UDINT;
	
	//
	FirstScan: BOOL:=TRUE;
END_VAR

                    
IF RestoreRetain THEN
	pApplication := CmpApp.AppFindApplicationByName('Application', ADR(ResultFind));
	ResultRestore := CmpApp.AppRestoreRetainsFromFile(pApplication, './Application/BackupRetain.ret');
	RestoreRetain := FALSE;
END_IF
   
IF SaveRetain THEN
	pApplication := CmpApp.AppFindApplicationByName('Application', ADR(ResultFind));
    ResultStore := AppStoreRetainsInFile(pApplication, './Application/BackupRetain.ret');
   	ResultStore := AppStoreRetainsInFile(pApplication, './Application/Application.ret');
   	SaveRetain := FALSE;
END_IF

// do not put anything below this
FirstScan := FALSE;
                  
END_PROGRAM

FUNCTION_BLOCK FB_DigitalOutput
VAR_INPUT
END_VAR
VAR_OUTPUT
END_VAR
VAR	
	// https://infosys.beckhoff.com/content/1033/tc3_plc_intro/11948825611.html?id=1756449079294237528
	Output AT %Q* : BOOL;
	_Output: BOOL;
	_FirstScan: BOOL;
END_VAR

                    IF _FirstScan THEN
	//
END_IF

// do some things?
Output :=_Output;

// do not put anything below this
_FirstScan := FALSE;
                  

METHOD PUBLIC Off : BOOL
VAR_INPUT
END_VAR
                          _Output := FALSE;
                        
END_METHOD

METHOD PUBLIC On : BOOL
VAR_INPUT
END_VAR
                          _Output := TRUE;
                        
END_METHOD

METHOD PUBLIC Toggle : BOOL
VAR_INPUT
END_VAR
                          _Output := NOT _Output;
                        
END_METHOD

{attribute 'monitoring' := 'variable'}
PROPERTY PUBLIC P_StateOff : BOOL
GET
VAR
END_VAR
                            P_StateOff := NOT _Output;
                          
END_GET
END_PROPERTY

{attribute 'monitoring' := 'variable'}
PROPERTY PUBLIC P_StateOn : BOOL
GET
VAR
END_VAR
                            P_StateOn := _Output;
                          
END_GET
END_PROPERTY
END_FUNCTION_BLOCK

FUNCTION F_ChangeJumpRow : BOOL
VAR_IN_OUT
	Command: DUT_Command;
END_VAR
VAR_INPUT
	BeginningRow: DINT;
	Change: INT;
END_VAR
VAR
	_LogicCmdParser : FB_ParseLogicCmd;
	_stLogicCmd : ST_LogicCmd;
END_VAR

                    // change the row that the jump function will jump to by the amount of the change
F_ChangeJumpRow := FALSE;
IF Command.CommandType = DUT_CommandType.LogicCommand THEN
	// parse the command string
	_LogicCmdParser(Command:=Command.CommandString, stCommand=>_stLogicCmd);
	
	// check the THEN function
	IF _stLogicCmd.THEN_Function = E_LogicFunction.JUMP AND_THEN _stLogicCmd.THEN_Function_Idx >= BeginningRow THEN
		_stLogicCmd.THEN_Function_Idx := _stLogicCmd.THEN_Function_Idx + Change;
		F_ChangeJumpRow := TRUE;
	END_IF
	
	// check the ELSE function
	IF _stLogicCmd.ELSE_Function = E_LogicFunction.JUMP AND_THEN _stLogicCmd.ELSE_Function_Idx >= BeginningRow  THEN
		_stLogicCmd.ELSE_Function_Idx := _stLogicCmd.ELSE_Function_Idx + Change;
		F_ChangeJumpRow := TRUE;
	END_IF
	
	// set the command
	IF F_ChangeJumpRow THEN
		Command.CommandString := F_BuildLogicCmd(stCommand:=_stLogicCmd);
	END_IF
	
ELSE
	F_ChangeJumpRow := FALSE;
	
END_IF
                  
END_FUNCTION

PROGRAM _20_Io
VAR
	//
	IoInputs: ARRAY [0..31] OF BYTE;
	IoOutputs: ARRAY [0..31] OF BYTE;
	
	//
	rx_heartbeat: BOOL;
	rx_en: BOOL;
    
    //
    IoOption: INT:=0;
	
	//
	FirstScan: BOOL:=TRUE;
END_VAR

                    //
IF FirstScan THEN
    //
END_IF

// leaving this pragma here for reference and for learning.
// it is not needed and was an attempt to parameterize configuring the IO
// the project define evaluates and could be a super handy technique in the future so I'll leave it here for reference.
// the defines for the project can be found in the Toolbar under Project -> Project Settings... -> Compile options -> Edit project defines...
{IF project_defined(IoOption1)}
    //IoOption := 1;
    //_M_MapIoOption1();
{ELSIF project_defined(IoOption2)}
    //IoOption := 2;
    //_M_MapIoOption2();
{ELSE}
    //IoOption := 0;
{END_IF}

// detect if the slave is connected and map its IO
IF IoOption1.wState = ETC_SLAVE_STATE.ETC_SLAVE_OPERATIONAL THEN
    _M_MapIoOption1();
END_IF
IF IoOption2.wState = ETC_SLAVE_STATE.ETC_SLAVE_OPERATIONAL THEN
    _M_MapIoOption2();
END_IF

// do not put anything below this
FirstScan := FALSE;
                  

METHOD PRIVATE _M_MapIoOption1
VAR_INPUT
END_VAR
                          // inputs
GVL.CmdIO.Input[0] := EL1809.Input_0;
GVL.CmdIO.Input[1] := EL1809.Input_1;
GVL.CmdIO.Input[2] := EL1809.Input_2;
GVL.CmdIO.Input[3] := EL1809.Input_3;
GVL.CmdIO.Input[4] := EL1809.Input_4;
GVL.CmdIO.Input[5] := EL1809.Input_5;
GVL.CmdIO.Input[6] := EL1809.Input_6;
GVL.CmdIO.Input[7] := EL1809.Input_7;
GVL.CmdIO.Input[8] := EL1809.Input_8;
GVL.CmdIO.Input[9] := EL1809.Input_9;
GVL.CmdIO.Input[10] := EL1809.Input_10;
GVL.CmdIO.Input[11] := EL1809.Input_11;
GVL.CmdIO.Input[12] := EL1809.Input_12;
GVL.CmdIO.Input[13] := EL1809.Input_13;
GVL.CmdIO.Input[14] := EL1809.Input_14;
GVL.CmdIO.Input[15] := EL1809.Input_15;

// outputs
EL2809.Output_0 := GVL.CmdIO.Output[0];
EL2809.Output_1 := GVL.CmdIO.Output[1];
EL2809.Output_2 := GVL.CmdIO.Output[2];
EL2809.Output_3 := GVL.CmdIO.Output[3];
EL2809.Output_4 := GVL.CmdIO.Output[4];
EL2809.Output_5 := GVL.CmdIO.Output[5];
EL2809.Output_6 := GVL.CmdIO.Output[6];
EL2809.Output_7 := GVL.CmdIO.Output[7];
EL2809.Output_8 := GVL.CmdIO.Output[8];
EL2809.Output_9 := GVL.CmdIO.Output[9];
EL2809.Output_10 := GVL.CmdIO.Output[10];
EL2809.Output_11 := GVL.CmdIO.Output[11];
EL2809.Output_12 := GVL.CmdIO.Output[12];
EL2809.Output_13 := GVL.CmdIO.Output[13];
EL2809.Output_14 := GVL.CmdIO.Output[14];
EL2809.Output_15 := GVL.CmdIO.Output[15];
                        
END_METHOD

METHOD PRIVATE _M_MapIoOption2
VAR_INST
	//
	TxCrc, RxCrc: UINT;
	ChecksumMisCount: INT;
	
	//
	HeartbeatOn: TON;
	HeartbeatOff: TON;
	HeartbeatPt: TIME:=T#1000MS;
    
    //
	bufferIdx: INT;
    
    //
    DeviceID: BYTE;
    IODeviceID: BYTE:=2;
	
END_VAR
                          //
HeartbeatOn(in:=NOT HeartbeatOff.Q,PT:=HeartbeatPt);
HeartbeatOff(in:=HeartbeatOn.Q,PT:=HeartbeatPt);


{region 'Output'}
// check that we are talking to the right device type
IF DeviceID = IODeviceID THEN
    // index 0 is for system outputs
    IoOutputs[0].0:=HeartbeatOn.Q; // send a heartbeat to the drive
    IoOutputs[0].1:=GVL.Enable; //
    // IoOutputs[0].2:=; //
    // IoOutputs[0].3:=; //
    // IoOutputs[0].4:=; //
    // IoOutputs[0].5:=; //
    // IoOutputs[0].6:=; //
    // IoOutputs[0].7:=; //
    
    // map outputs
    IoOutputs[1].0 := GVL.CmdIO.Output[0];
    IoOutputs[1].1 := GVL.CmdIO.Output[1];
    IoOutputs[1].2 := GVL.CmdIO.Output[2];
    IoOutputs[1].3 := GVL.CmdIO.Output[3];
    IoOutputs[1].4 := GVL.CmdIO.Output[4];
    IoOutputs[1].5 := GVL.CmdIO.Output[5];
    IoOutputs[1].6 := GVL.CmdIO.Output[6];
    IoOutputs[1].7 := GVL.CmdIO.Output[7];
    IoOutputs[2].0 := GVL.CmdIO.Output[8];
    IoOutputs[2].1 := GVL.CmdIO.Output[9];
    IoOutputs[2].2 := GVL.CmdIO.Output[10];
    IoOutputs[2].3 := GVL.CmdIO.Output[11];
    IoOutputs[2].4 := GVL.CmdIO.Output[12];
    IoOutputs[2].5 := GVL.CmdIO.Output[13];
    IoOutputs[2].6 := GVL.CmdIO.Output[14];
    IoOutputs[2].7 := GVL.CmdIO.Output[15];
    
    // bytes 3 through 28 are unused
    //
    
    // byte 29 will be used to send the expected device id
    IoOutputs[29] := IODeviceID;
    
END_IF

// bytes 30 and 31 will be used for crc
// calc crc here
TxCrc := F_Checksum(ADR(IoOutputs), 30);
// append calc crc to tx buffer
MEMUtils.MemCpy(pbyDest:=ADR(IoOutputs[30]), 
				pbySrc:=ADR(TxCrc), 
				dwSize:=2);
{endregion}
	
{region 'Input'}
// copy crc from rx buffer
MEMUtils.MemCpy(pbyDest:=ADR(RxCrc), 
				pbySrc:=ADR(IoInputs[30]), 
				dwSize:=2);

// compare calc crc with rx crc
IF RxCrc = F_Checksum(ADR(IoInputs), 30) THEN
	// byte 0 is for system inputs
	rx_heartbeat	:= IoInputs[0].0; // receive the heartbeat back
	rx_en 			:= IoInputs[0].1; // receive the enable back
	//	 			:= IoInputs[0].2;
	// 				:= IoInputs[0].3;
	// 				:= IoInputs[0].4;
	// 				:= IoInputs[0].5;
	// 				:= IoInputs[0].6;
	// 				:= IoInputs[0].7;
    
    // map inputs
    GVL.CmdIO.Input[0] := IoInputs[1].0;
    GVL.CmdIO.Input[1] := IoInputs[1].1;
    GVL.CmdIO.Input[2] := IoInputs[1].2;
    GVL.CmdIO.Input[3] := IoInputs[1].3;
    GVL.CmdIO.Input[4] := IoInputs[1].4;
    GVL.CmdIO.Input[5] := IoInputs[1].5;
    GVL.CmdIO.Input[6] := IoInputs[1].6;
    GVL.CmdIO.Input[7] := IoInputs[1].7;
    GVL.CmdIO.Input[8] := IoInputs[2].0;
    GVL.CmdIO.Input[9] := IoInputs[2].1;
    GVL.CmdIO.Input[10] := IoInputs[2].2;
    GVL.CmdIO.Input[11] := IoInputs[2].3;
    GVL.CmdIO.Input[12] := IoInputs[2].4;
    GVL.CmdIO.Input[13] := IoInputs[2].5;
    GVL.CmdIO.Input[14] := IoInputs[2].6;
    GVL.CmdIO.Input[15] := IoInputs[2].7;
	
	// bytes 3 through 28 are unused
	//
    
    // byte 29 will be used to identify the device
	DeviceID := IoInputs[29];
	
	// Rx buffer index 30 and 31 will be for crc
ELSE
	// increment crc mismatch counter
	ChecksumMisCount := ChecksumMisCount + 1;
END_IF
{endregion}
                        
END_METHOD
END_PROGRAM

FUNCTION F_RadToDeg : LREAL
VAR_INPUT
    Radians: LREAL;
END_VAR
VAR
END_VAR

                    F_RadToDeg := Radians * (180 / GVL.pi);
                  
END_FUNCTION

PROGRAM _60_PathPlanner
VAR
	PlanPath: FB_CncPathPlanner;
END_VAR
VAR CONSTANT
	wVarCount : WORD := 1;
END_VAR
VAR
	lrR1 : LREAL:=30;
	
	astVar : ARRAY [0..wVarCount] OF SMC_SingleVar :=
			[(strVarName:='R1', pAdr := ADR(lrR1), eVarType := SMC_VarType.SMC_TYPE_LREAL)];
			
	stVarList : SMC_VarList := (wNumberVars := wVarCount, psvVarlist := ADR(astVar));
END_VAR

                    // this has to be called in a separate task with lower priority
// https://content.helpme-codesys.com/en/libs/SM3_CNC/Current/SM_CNC_POUs/NC2/Interpreter/SMC_NCInterpreter.html
PlanPath(VarList:= stVarList, DataOut=> );
                  
END_PROGRAM

(* Round LREAL to nearest INT (half away from zero via ±0.5 then truncate).
   LREAL_TO_INT alone truncates toward zero (27.8->27, -27.8->-27), which
   systematically under-drives |Hz| and biases crawl toward stop.
   Positive: add 0.5 then LREAL_TO_INT. Negative: subtract 0.5 then LREAL_TO_INT
   so both sides round to nearest (e.g. 27.8->28, -27.8->-28).
   Used when converting LREAL step rate (Hz) to INT16 for the Teensy PTO. *)

FUNCTION F_RoundToInt : INT
VAR_INPUT
	x : LREAL;
END_VAR
VAR
END_VAR

                    IF x >= 0.0 THEN
    F_RoundToInt := LREAL_TO_INT(x + 0.5);
ELSE
    F_RoundToInt := LREAL_TO_INT(x - 0.5);
END_IF
                  
END_FUNCTION

FUNCTION_BLOCK FB_LicenseStatus IMPLEMENTS CmpEventMgr.ICmpEventCallback
VAR_OUTPUT
	eState : CmpMgr.RUNTIME_LICENSE_STATE;
	udiSecondsLeft : UDINT;
	udiMinutesLeft : UDINT;
	tRemaining : TIME;
	sState : STRING(32);
	sBanner : STRING(80);
	xDemo : BOOL;
	xLicensed : BOOL;
	xShowBanner : BOOL;
END_VAR
VAR
	_hEvent : SysTypes.RTS_IEC_HANDLE := SysTypes.RTS_INVALID_HANDLE;
	_hCallback : SysTypes.RTS_IEC_HANDLE := SysTypes.RTS_INVALID_HANDLE;
	_result : SysTypes.RTS_IEC_RESULT;
	_xRegistered : BOOL;
	_xTried : BOOL;
	_xGotEvent : BOOL;
	_udiSecondsAtEvent : UDINT;
	_tEvent : TIME;
	_tRetry : TIME;
	_udiElapsed : UDINT;
	_sMin : STRING(11);
	_sSec : STRING(11);
	_udiSec : UDINT;
END_VAR

                    M_EnsureRegistered();
M_UpdateRemaining();
M_BuildBanner();
                  

METHOD EventCallback : SysTypes.RTS_IEC_RESULT
VAR_INPUT
	pEventParam : POINTER TO CmpEventMgr.EventParam;
END_VAR
VAR
	pLic : POINTER TO CmpMgr.EVTPARAM_CmpMgr_LicenseState;
END_VAR
                          EventCallback := 0;
IF pEventParam = 0 THEN
	RETURN;
END_IF
IF pEventParam^.EventId <> CmpMgr.EventIDs.EVT_CmpMgr_LicenseState THEN
	RETURN;
END_IF
IF pEventParam^.pParameter = 0 THEN
	RETURN;
END_IF

pLic := pEventParam^.pParameter;
eState := pLic^.state;
_xGotEvent := TRUE;
_tEvent := TIME();
IF pLic^.secondsToExpiration > 0 THEN
	_udiSecondsAtEvent := pLic^.secondsToExpiration;
ELSIF eState = CmpMgr.RUNTIME_LICENSE_STATE.DEMOMODE THEN
	_udiSecondsAtEvent := 7200;
ELSE
	_udiSecondsAtEvent := 0;
END_IF
udiSecondsLeft := _udiSecondsAtEvent;
                        
END_METHOD

METHOD FB_Init : BOOL
VAR_INPUT
	bInitRetains : BOOL;
	bInCopyCode : BOOL;
END_VAR
                          IF NOT bInCopyCode THEN
	M_EnsureRegistered();
END_IF
FB_Init := TRUE;
                        
END_METHOD

METHOD FB_Exit : BOOL
VAR_INPUT
	bInCopyCode : BOOL;
END_VAR
                          IF NOT bInCopyCode THEN
	M_Unregister();
END_IF
FB_Exit := TRUE;
                        
END_METHOD

METHOD PRIVATE M_EnsureRegistered
VAR
	tNow : TIME;
END_VAR
                          IF _xRegistered THEN
	RETURN;
END_IF

tNow := TIME();
IF _xTried AND ((tNow - _tRetry) < T#2S) THEN
	RETURN;
END_IF
_xTried := TRUE;
_tRetry := tNow;

IF _hEvent = SysTypes.RTS_INVALID_HANDLE THEN
	_hEvent := CmpEventMgr.EventOpen(
		EventId := CmpMgr.EventIDs.EVT_CmpMgr_LicenseState,
		CmpIdProvider := CmpMgr.ComponentID.CMPID_CmpMgr,
		Result := _result);
END_IF

IF _hEvent = SysTypes.RTS_INVALID_HANDLE THEN
	RETURN;
END_IF

_hCallback := CmpEventMgr.EventRegisterCallback2(
	hEvent := _hEvent,
	pICallback := THIS^,
	pUserParameter := 0,
	Result := _result);

IF _hCallback <> SysTypes.RTS_INVALID_HANDLE THEN
	_xRegistered := TRUE;
END_IF
                        
END_METHOD

